		CASE FC OF
		(******************************************************************)
		1..2: (* 0x01 Read Coil Status , 0x02 Read Input Status *)
			IF R_POINTS <= 2000 THEN
				w_tmp := INT_TO_WORD(R_ADDR);
				S_BUF.BUFFER[08] := WORD_TO_BYTE(SHR(w_tmp,8));
				S_BUF.BUFFER[09] := WORD_TO_BYTE(w_tmp);
				w_tmp := INT_TO_WORD(R_POINTS);
				S_BUF.BUFFER[10] := WORD_TO_BYTE(SHR(w_tmp,8));
				S_BUF.BUFFER[11] := WORD_TO_BYTE(w_tmp);
				S_BUF.SIZE := UINT#12;
				Response :=	WORD_TO_INT(SHR(INT_TO_WORD(R_POINTS + 7),3));
				comp := 7;
			ELSE
				ERROR := DWORD#2; (* ILLEGAL DATA ADDRESS *)
			END_IF;
		(******************************************************************)
		3..4: (* 0x03 Read Holding Registers , 0x04 Read Input Registers *)
			IF R_POINTS <= 125 THEN
				w_tmp := INT_TO_WORD(R_ADDR);
				S_BUF.BUFFER[08] := WORD_TO_BYTE(SHR(w_tmp,8));
				S_BUF.BUFFER[09] := WORD_TO_BYTE(w_tmp);
				w_tmp := INT_TO_WORD(R_POINTS);
				S_BUF.BUFFER[10] := WORD_TO_BYTE(SHR(w_tmp,8));
				S_BUF.BUFFER[11] := WORD_TO_BYTE(w_tmp);
				S_BUF.SIZE := UINT#12;
				Response :=	WORD_TO_INT(SHL(w_tmp,1));
				comp := 7;
			ELSE
				ERROR := DWORD#2; (* ILLEGAL DATA ADDRESS *)
			END_IF;
		(******************************************************************)
		5:	(* 0x05 Force Single Coil *)
			IF W_DATA_ADR <= DATA_SIZE THEN
				w_tmp := INT_TO_WORD(W_ADDR);
				S_BUF.BUFFER[08] := WORD_TO_BYTE(SHR(w_tmp,8));
				S_BUF.BUFFER[09] := WORD_TO_BYTE(w_tmp);
				S_BUF.BUFFER[10] := SEL((DATA[W_DATA_ADR] AND SHL(WORD#1,W_DATA_BITPOS))>WORD#00,BYTE#16#00,BYTE#16#FF);
				S_BUF.BUFFER[11] := BYTE#00;
				S_BUF.SIZE := UINT#12;
				Response := 3;
				comp := 11;
			ELSE
				ERROR := DWORD#2; (* ILLEGAL DATA ADDRESS *)
			END_IF;
		(******************************************************************)
		6:	(* 0x06 Preset Single Register *)
			IF W_DATA_ADR <= DATA_SIZE THEN
				w_tmp := INT_TO_WORD(W_ADDR);
				S_BUF.BUFFER[08] := WORD_TO_BYTE(SHR(w_tmp,8));
				S_BUF.BUFFER[09] := WORD_TO_BYTE(w_tmp);
				w_tmp := DATA[W_DATA_ADR];
				S_BUF.BUFFER[10] := WORD_TO_BYTE(SHR(w_tmp,8));
				S_BUF.BUFFER[11] := WORD_TO_BYTE(w_tmp);
				S_BUF.SIZE := UINT#12;
				Response := 3;
				comp := 11;
			ELSE
				ERROR := DWORD#2; (* ILLEGAL DATA ADDRESS *)
			END_IF;
		(******************************************************************)
		15:	(* 0x0F Force Multiple Coils *)
			IF (WORD_TO_INT(SHR(INT_TO_WORD(WORD_TO_INT(SHL(INT_TO_WORD(W_DATA_ADR),4)) + W_POINTS + W_DATA_BITPOS + 15),4)) <= DATA_SIZE) AND W_POINTS <= 1968 THEN
				w_tmp := INT_TO_WORD(W_ADDR);
				S_BUF.BUFFER[08] := WORD_TO_BYTE(SHR(w_tmp,8));
				S_BUF.BUFFER[09] := WORD_TO_BYTE(w_tmp);
				w_tmp := INT_TO_WORD(W_POINTS);
				S_BUF.BUFFER[10] := WORD_TO_BYTE(SHR(w_tmp,8));
				S_BUF.BUFFER[11] := WORD_TO_BYTE(w_tmp);
				S_BUF.BUFFER[12] := WORD_TO_BYTE(SHR(INT_TO_WORD(W_POINTS + 7),3));

				w_mask := SHL(WORD#1,W_DATA_BITPOS);
				bit_pos := 0;
				w_tmp := WORD#00;
				idx1 := 12;
				idx2 := W_DATA_ADR;
				FOR i := 1 TO W_POINTS DO
					w_tmp :=OSCAT_BASIC.BIT_LOAD_W(w_tmp,(DATA[idx2] AND w_mask) > WORD#0,bit_pos);
					bit_pos := bit_pos + 1;
					IF bit_pos > 7 OR i=W_POINTS THEN
						bit_pos := 0;
						idx1 := idx1 + 1;
						S_BUF.BUFFER[idx1] := WORD_TO_BYTE(w_tmp);
						w_tmp := WORD#0;
					END_IF;
					w_mask := ROL(w_mask,1);
					IF w_mask = WORD#1 THEN
						idx2 := idx2 +1;
					END_IF;
				END_FOR;
				S_BUF.SIZE := INT_TO_UINT(idx1 + 1);
				Response := 3;
				comp := 11;
			ELSE
				ERROR := DWORD#2; (* ILLEGAL DATA ADDRESS *)
			END_IF;
		(******************************************************************)
		16:	(* 0x10 Write Multiple Registers *)
			IF W_DATA_ADR + W_POINTS <= DATA_SIZE AND W_POINTS <= 123 THEN
				w_tmp := INT_TO_WORD(W_ADDR);
				S_BUF.BUFFER[08] := WORD_TO_BYTE(SHR(w_tmp,8));
				S_BUF.BUFFER[09] := WORD_TO_BYTE(w_tmp);
				w_tmp := INT_TO_WORD(W_POINTS);
				S_BUF.BUFFER[10] := WORD_TO_BYTE(SHR(w_tmp,8));
				S_BUF.BUFFER[11] := WORD_TO_BYTE(w_tmp);
				S_BUF.BUFFER[12] := SHL(S_BUF.BUFFER[11],1);
			
				idx1 := 11;
				count := W_DATA_ADR + W_POINTS - 1;
				FOR i := W_DATA_ADR TO count DO
					idx1 := idx1 + 2;
					idx2 := idx1 + 1; (* zweiter index für pcworx notwendig ! *)
					w_tmp := DATA[i];
					S_BUF.BUFFER[idx1] := WORD_TO_BYTE(SHR(w_tmp,8));
					S_BUF.BUFFER[idx2] := WORD_TO_BYTE(w_tmp);
				END_FOR;

				S_BUF.SIZE := INT_TO_UINT(idx2 + 1);
				Response := 3;
				comp := 11;
			ELSE
				ERROR := DWORD#2; (* ILLEGAL DATA ADDRESS *)
			END_IF;
		(******************************************************************)
		22:	(* 0x16 Mask Write Register *)
			IF W_DATA_ADR + 2 <= DATA_SIZE THEN
				w_tmp := INT_TO_WORD(W_ADDR);
				S_BUF.BUFFER[08] := WORD_TO_BYTE(SHR(w_tmp,8));
				S_BUF.BUFFER[09] := WORD_TO_BYTE(w_tmp);
				idx1 := W_DATA_ADR;
				w_tmp := DATA[idx1];
				S_BUF.BUFFER[10] := WORD_TO_BYTE(SHR(w_tmp,8));
				S_BUF.BUFFER[11] := WORD_TO_BYTE(w_tmp);
				idx1 := idx1 +1;
				w_tmp := DATA[idx1];
				S_BUF.BUFFER[12] := WORD_TO_BYTE(SHR(w_tmp,8));
				S_BUF.BUFFER[13] := WORD_TO_BYTE(w_tmp);

				S_BUF.SIZE := UINT#14;
				Response := 5;
				comp := 13;
			ELSE
				ERROR := DWORD#2; (* ILLEGAL DATA ADDRESS *)
			END_IF;
		(******************************************************************)
		23:	(* 0x17 Read/Write Multible Registers *)
			IF W_DATA_ADR + W_POINTS <= DATA_SIZE AND W_POINTS <= 121 AND R_POINTS <= 125 THEN
				idx1 := 15;
				count := W_DATA_ADR + W_POINTS - 1;
				FOR i := W_DATA_ADR TO count DO
					idx1 := idx1 + 2;
					idx2 := idx1 + 1; (* zweiter index für pcworx notwendig ! *)
					w_tmp := DATA[i];
					S_BUF.BUFFER[idx1] := WORD_TO_BYTE(SHR(w_tmp,8));
					S_BUF.BUFFER[idx2] := WORD_TO_BYTE(w_tmp);
				END_FOR;

				(* WRITE *)
				w_tmp := INT_TO_WORD(W_ADDR);
				S_BUF.BUFFER[12] := WORD_TO_BYTE(SHR(w_tmp,8));
				S_BUF.BUFFER[13] := WORD_TO_BYTE(w_tmp);
				w_tmp := INT_TO_WORD(W_POINTS);
				S_BUF.BUFFER[14] := WORD_TO_BYTE(SHR(w_tmp,8));
				S_BUF.BUFFER[15] := WORD_TO_BYTE(w_tmp);
				S_BUF.BUFFER[16] := SHL(S_BUF.BUFFER[15],1);

				(* READ *)
				w_tmp := INT_TO_WORD(R_ADDR);
				S_BUF.BUFFER[08] := WORD_TO_BYTE(SHR(w_tmp,8));
				S_BUF.BUFFER[09] := WORD_TO_BYTE(w_tmp);
				w_tmp := INT_TO_WORD(R_POINTS);
				S_BUF.BUFFER[10] := WORD_TO_BYTE(SHR(w_tmp,8));
				S_BUF.BUFFER[11] := WORD_TO_BYTE(w_tmp);

				S_BUF.SIZE := INT_TO_UINT(idx2 + 1);
				Response := WORD_TO_INT(SHL(w_tmp,1));
				comp := 7;
			ELSE
				ERROR := DWORD#2; (* ILLEGAL DATA ADDRESS *)
			END_IF;
		(******************************************************************)

		ELSE
			ERROR := DWORD#00000001; (* ILLEGAL FUNCTION *)
		END_CASE;

		(* Daten senden *)
		IF ERROR = DWORD#00 THEN
			Transaction_ID := Transaction_ID + 1;
			w_tmp := UINT_TO_WORD(S_BUF.SIZE - UINT#6);
			(* ---- H E A D E R --------------------------------------------------------------- *)
			S_BUF.BUFFER[0] := IP_ID; (* TRANSACTION-ID HI-Byte *)
			S_BUF.BUFFER[1] := INT_TO_BYTE(Transaction_ID); (* TRANSACTION-ID LO-Byte *)
			S_BUF.BUFFER[2] := BYTE#00; (* PROTOKOLL-ID HI-Byte *)
			S_BUF.BUFFER[3] := BYTE#00; (* PROTOKOLL-ID LO-Byte *)
			S_BUF.BUFFER[4] := WORD_TO_BYTE(SHR(w_tmp,8)); (* Laenge HI-Byte *)
			S_BUF.BUFFER[5] := WORD_TO_BYTE(w_tmp); (* Laenge LO-Byte *)
			S_BUF.BUFFER[6] := UNIT_ID; (* UNIT *)
			S_BUF.BUFFER[7] := INT_TO_BYTE(FC); (* FUNCTION-CODE *)
			(*----- END OF HEADER --------------------------------------------------------------*)
			R_BUF.SIZE := UINT#0; (* Empfangsbuffer löschen *)
			state := 30; (* wait for response *)
		ELSE
			IP_STATE := BYTE#4; (* Abmelden *)
			state := 00;
		END_IF;
	END_IF;

30: (* response *)
	IF IP_C.ERROR <> DWORD#00 THEN
		ERROR := IP_C.ERROR;
		IP_STATE := BYTE#4; (* Abmelden *)
		state := 00;
	ELSIF S_BUF.SIZE = UINT#0 AND R_BUF.SIZE > UINT#0 THEN
		(* erwartete länge in sendebuffer nachträglich eintragen um vergleich zu ermöglichen *)
		w_tmp := INT_TO_WORD(Response + 3);
		S_BUF.BUFFER[4] := WORD_TO_BYTE(SHR(w_tmp,8));
		S_BUF.BUFFER[5] := WORD_TO_BYTE(w_tmp);

		FOR i := 0 TO comp DO
			IF S_BUF.BUFFER[i] <> R_BUF.BUFFER[i] THEN EXIT; END_IF;
		END_FOR;

		IF R_BUF.SIZE >= UINT#9 AND R_BUF.BUFFER[7] > BYTE#128 THEN  (* Bit 7 = Error Message *)
			ERROR := BYTE_TO_DWORD(R_BUF.BUFFER[8]);
			IP_STATE := BYTE#4; (* Abmelden *)
			state := 00;
		ELSIF R_BUF.SIZE = INT_TO_UINT(Response + 9) AND i > comp THEN
			mask := SHL(DWORD#1,FC);
			(* READ_COILS, READ_INPUT_DISCRETES *)
			IF (mask AND DWORD#2#00000000_00000000_00000000_00000110) > DWORD#0 THEN (* FC 1,2 *)
				IF WORD_TO_INT(SHR(INT_TO_WORD(WORD_TO_INT(SHL(INT_TO_WORD(R_DATA_ADR),4)) + R_POINTS + R_DATA_BITPOS + 15),4)) <= DATA_SIZE THEN
					b_mask := BYTE#1;
					idx1 := 09;
					idx2 := R_DATA_ADR;
					bit_pos := R_DATA_BITPOS;
					FOR i := 1 TO R_POINTS DO
						DATA[idx2]:=OSCAT_BASIC.BIT_LOAD_W(DATA[idx2],(R_BUF.BUFFER[idx1] AND b_mask) > BYTE#0,bit_pos);
						bit_pos := bit_pos + 1;
						IF bit_pos > 15 THEN
							idx2 := idx2 + 1;
							bit_pos := 0;
						END_IF;
						b_mask := ROL(b_mask,1);
						IF b_mask = BYTE#1 THEN
							idx1 := idx1 + 1;
						END_IF;
					END_FOR;
				ELSE
					ERROR := DWORD#2; (* ILLEGAL DATA ADDRESS *)
				END_IF;

			(* READ_MULTIPLE_REGISTERS, READ_INPUT_REGISTERS, READ_WRITE_REGISTERS *)
			ELSIF (mask AND DWORD#2#00000000_10000000_00000000_00011000) > DWORD#0 THEN (* FC 3,4,23 *)
				IF R_DATA_ADR + R_POINTS <= DATA_SIZE THEN
					stop := R_DATA_ADR + R_POINTS -1 ;
					idx1 := 07;
					FOR i := R_DATA_ADR TO stop DO
						idx1 := idx1 + 2;
						idx2 := idx1 + 1;
						DATA[i] := OSCAT_BASIC.WORD_OF_BYTE(R_BUF.BUFFER[idx1],R_BUF.BUFFER[idx2]);
					END_FOR;
				ELSE
					ERROR := DWORD#2; (* ILLEGAL DATA ADDRESS *)
				END_IF;
			ELSIF (mask AND DWORD#2#11111111_00111110_01111111_10000001) > DWORD#0 THEN (* ILLEGAL FUNCTION CODE ? *)
				ERROR := DWORD#1; (* ILLEGAL FUNCTION *)
			END_IF;
		ELSE
			ERROR := DWORD#3; (* ILLEGAL DATA VALUE *)
		END_IF;

		IP_STATE := BYTE#4; (* Abmelden *)
		state := 00;
		R_BUF.SIZE := UINT#0;

	END_IF;

END_CASE;

(* IP_FIFO *)
IP_FIFO(FIFO:=IP_C.FIFO,STATE:=IP_STATE,ID:=IP_ID);
BUSY := IP_STATE = BYTE#3;

(* revision history
ks	05. jan. 2009	rev 1.0
	original version

ks	28. jan. 2009	rev 1.1
	network_buffer_short verwendet  

ks	20. oct. 2009	rev 1.2
Networkbuffer und Buffer-funktionen auf Basis 0

*)

END_FUNCTION_BLOCK

// POUs/NETWORK/MB_SERVER
FUNCTION_BLOCK MB_SERVER
VAR_IN_OUT
	IP_C : IP_C;
	S_BUF : NETWORK_BUFFER_SHORT;
	R_BUF : NETWORK_BUFFER_SHORT;
	VMAP : ARRAY [1..10] OF VMAP_DATA;
	DATA : ARRAY [0..255] OF WORD;
END_VAR
VAR_INPUT
	DATA_SIZE : INT;
	ENABLE : BOOL;
	UDP : BOOL;
END_VAR
VAR_OUTPUT
	ERROR : DWORD;
END_VAR
VAR
	MB_VMAP : MB_VMAP;
	adr1 : INT;
	adr2 : INT;
	points : INT;
	points2 : INT;
	coils : BYTE;
	mask : BYTE;
	idx1 : INT;
	idx2 : INT;
	bit_pos : INT;
	count : INT;
	fc : INT;
	i : INT;
	state : INT;
	ip_state : BYTE;
	ip_id : BYTE;
	IP_FIFO : IP_FIFO;
	w_tmp : WORD;
	last_cycle : TIME;
	tx : TIME;
	t : TON;
	ip_error : BOOL;
END_VAR

(*

version 1.4		05. may. 2012
programmer 		ks
tested by		ks

MB_SERVER ermöglicht das Lesen/Schreiben von Daten durch ein Remote-Device mittels Modbus over Ethernet (OpenModbus)

*)

(* read system time *)
tx := DWORD_TO_TIME(OSCAT_BASIC.T_PLC_MS());

FOR i := 1 TO 10 DO
	IF VMAP[i].TIME_OUT > T#0s THEN
		VMAP[i].TIME_OUT := VMAP[i].TIME_OUT + tx - last_cycle;
	END_IF;
END_FOR;
last_cycle := tx;
ip_error := IP_C.ERROR > DWORD#0;

CASE state OF
00: (* Warten auf Freigabe *)
	IF ENABLE THEN
		state := 10;
		ip_state := BYTE#1; (* Anmelden *)
	END_IF;

10: (* Bei IP_Control anmelden und auf freigabe warten *)
	IF ip_state = BYTE#3 THEN

		(* IP Datenverkehr einrichten *)
		IP_C.C_PORT := WORD#0; (* Port von IP_CONTROL verwenden *)
		IP_C.C_IP := DWORD#0; (* IP von IP_CONTROL verwenden *)
		IP_C.C_MODE := SEL(UDP,BYTE#4,BYTE#5); (* Mode: 4=TCP+PASSIV+PORT , 5=UDP+PASSIV+PORT *)
		IP_C.TIME_RESET := TRUE; (* Zeitueberwachung rücksetzen *)
		IP_C.C_ENABLE := TRUE; (* Verbindungsaufbau freigeben *)
		IP_C.R_OBSERVE := TRUE; (* keine Empfangsueberwachung *)
		state := 20;
	END_IF;

20:	IF NOT ip_error THEN
		IF S_BUF.SIZE = UINT#0 AND R_BUF.SIZE > UINT#6 THEN	(* Datensenden nicht aktiv und Daten wurden empfangen *)
			IF  R_BUF.SIZE = WORD_TO_UINT(OSCAT_BASIC.WORD_OF_BYTE(R_BUF.BUFFER[4],R_BUF.BUFFER[5])) + UINT#6 THEN (* gültige Datenlänge *)
				ERROR := DWORD#00; (* Error löschen *)

				(* Header kopieren *)
				FOR i := 0 TO 13 DO
					S_BUF.BUFFER[i] := R_BUF.BUFFER[i];
				END_FOR;
				fc := BYTE_TO_INT(R_BUF.BUFFER[7]);
				adr1 := WORD_TO_INT(OSCAT_BASIC.WORD_OF_BYTE(R_BUF.BUFFER[8],R_BUF.BUFFER[9]));
				points := WORD_TO_INT(OSCAT_BASIC.WORD_OF_BYTE(R_BUF.BUFFER[10],R_BUF.BUFFER[11]));

				(* Virtual Address *)
				MB_VMAP(VMAP:=VMAP,FC:=fc,V_ADR:=adr1,V_CNT:=points,SIZE:=DATA_SIZE);
				adr1:=MB_VMAP.P_ADR;
				bit_pos:=MB_VMAP.P_BIT;
				ERROR:=BYTE_TO_DWORD(MB_VMAP.ERROR);

				IF ERROR = DWORD#0 THEN
					CASE fc OF
					(*---------------------------------------------*)
					1..2 : (* Read Coil Status / Read Input Status *)
						count := 9; (* erstes Datenbyte *)
						coils := BYTE#0;
						mask := BYTE#1;
						FOR i := 1 TO points DO
							IF mask = BYTE#0 THEN
								mask := BYTE#1;
								S_BUF.BUFFER[count] := coils;
								coils := BYTE#0;
								count := count + 1;
							END_IF;
							IF (DATA[adr1] AND SHL(WORD#1,bit_pos)) > WORD#0 THEN
								coils := coils OR mask;
							END_IF;
	
							bit_Pos := bit_Pos + 1;
							IF bit_pos > 15 THEN
								ADR1 := ADR1 + 1;
								bit_pos := 0;
							END_IF;
	
							mask := SHL(mask,1);
						END_FOR;
						S_BUF.BUFFER[Count] := coils;
	
						S_BUF.BUFFER[8] := INT_TO_BYTE(count - 8); (* Bytecount *)
						S_BUF.SIZE := INT_TO_UINT(count + 1);
	
					(*--------------------------------------------------*)
					3..4 : (* Read Holding Registers / Read Input Registers *)
						idx1 := 07;
						count := adr1 + points - 1;
						FOR i := adr1 TO count DO
							idx1 := idx1 + 2;
							idx2 := idx1 + 1; (* zweiter index für pcworx notwendig ! *)
							w_tmp := DATA[i];
							S_BUF.BUFFER[idx1] := WORD_TO_BYTE(SHR(w_tmp,8));
							S_BUF.BUFFER[idx2] := WORD_TO_BYTE(w_tmp);
						END_FOR;
						S_BUF.BUFFER[8] := SHL(INT_TO_BYTE(points),1); (* Anzahl Register in Bytes *)
						S_BUF.SIZE := INT_TO_UINT(idx2 + 1);
					(*--------------------------------------------------*)
					5 : (* Force Single Coil *)
						DATA[adr1]:=OSCAT_BASIC.BIT_LOAD_W(DATA[adr1],R_BUF.BUFFER[10] > BYTE#0,bit_pos);
						S_BUF.SIZE := UINT#12;
					(*--------------------------------------------------*)
					6 : (* Preset Single Register *)
						DATA[adr1] := OSCAT_BASIC.WORD_OF_BYTE(R_BUF.BUFFER[10],R_BUF.BUFFER[11]);
						S_BUF.SIZE := UINT#12;
					(*--------------------------------------------------*)
					15 : (* Force Multible Coils *)
						mask := BYTE#1;
						idx1 := 13;
						FOR i := 1 TO points DO
							DATA[adr1]:=OSCAT_BASIC.BIT_LOAD_W(DATA[adr1],(R_BUF.BUFFER[idx1] AND mask) > BYTE#0,bit_pos);
							bit_pos := bit_pos + 1;
							IF bit_pos > 15 THEN
								adr1:= adr1 + 1;
								bit_pos := 0;
							END_IF;
							mask := ROL(mask,1);
							IF mask = BYTE#1 THEN
								idx1 := idx1 +1;
							END_IF;
						END_FOR;
						S_BUF.SIZE := UINT#12;
					(*--------------------------------------------------*)
					16 : (* Preset Multiple Registers	*)
						idx1 := 11;
						count := adr1 + points - 1;
						FOR i := adr1 TO Count DO
							idx1 := idx1 + 2;
	 						idx2 := idx1 + 1;
							Data[i] := OSCAT_BASIC.WORD_OF_BYTE(R_BUF.BUFFER[idx1],R_BUF.BUFFER[idx2]);
						END_FOR;
						S_BUF.SIZE := UINT#12;
					(*--------------------------------------------------*)
					22 : (* Mask Write Register *)
						w_tmp := OSCAT_BASIC.WORD_OF_BYTE(R_BUF.BUFFER[10],R_BUF.BUFFER[11]); (* and mask *)
						DATA[adr1] := (DATA[adr1] AND w_tmp) OR (OSCAT_BASIC.WORD_OF_BYTE(R_BUF.BUFFER[12],R_BUF.BUFFER[13]) AND (NOT w_tmp));
						S_BUF.SIZE := UINT#14;
					(*--------------------------------------------------*)
					23 : (* Read / Write Registers	*)
						(*--- Write-Register -----------------------------------*)
						adr2 := WORD_TO_INT(OSCAT_BASIC.WORD_OF_BYTE(R_BUF.BUFFER[12],R_BUF.BUFFER[13]));
						points2 := WORD_TO_INT(OSCAT_BASIC.WORD_OF_BYTE(R_BUF.BUFFER[14],R_BUF.BUFFER[15]));

						(* Virtual Address Write Register *)
						MB_VMAP(VMAP:=VMAP,FC:=16,V_ADR:=adr2,V_CNT:=points2,SIZE:=DATA_SIZE);
						adr2:=MB_VMAP.P_ADR;
						ERROR:=BYTE_TO_DWORD(MB_VMAP.ERROR);
	
						IF ERROR = DWORD#0 THEN
							idx1 := 15;
							count := adr2 + points2 - 1;
							FOR i := adr2 TO count DO
								idx1 := idx1 + 2;
	 							idx2 := idx1 + 1; (* zweiter index für pcworx notwendig ! *)
								Data[i] := OSCAT_BASIC.WORD_OF_BYTE(R_BUF.BUFFER[idx1],R_BUF.BUFFER[idx2]);
							END_FOR;
	
							(*--- Read-Register -----------------------------------*)
							idx1 := 07;
							count := adr1 + points - 1;
							FOR i := adr1 TO count DO
								idx1 := idx1 + 2;
								idx2 := idx1 + 1; (* zweiter index für pcworx notwendig ! *)
								w_tmp := DATA[i];
								S_BUF.BUFFER[idx1] := WORD_TO_BYTE(SHR(w_tmp,8));
								S_BUF.BUFFER[idx2] := WORD_TO_BYTE(w_tmp);
							END_FOR;
							S_BUF.BUFFER[8] := SHL(INT_TO_BYTE(points),1); (* Anzahl Register in Bytes *)
							S_BUF.SIZE := INT_TO_UINT(idx2 + 1);
	
						END_IF;
	
					(*--------------------------------------------------*)
					ELSE
						ERROR := DWORD#01; (* ILLEGAL FUNCTION *)
					END_CASE;
				END_IF;
			END_IF;
	
			IF ERROR > DWORD#0 THEN
				S_BUF.BUFFER[7] := S_BUF.BUFFER[7] OR BYTE#2#1000_0000; (* Fehlerbit setzen *)
				S_BUF.BUFFER[8] := DWORD_TO_BYTE(ERROR);
				S_BUF.SIZE := UINT#9;
			END_IF;
	
			S_BUF.BUFFER[4] := BYTE#0; (* high Byte *)
			S_BUF.BUFFER[5] := UINT_TO_BYTE(S_BUF.SIZE - UINT#6); (* Längenfeld eintragen - nur low byte *)
	
		END_IF;
	ELSE
		ERROR := IP_C.ERROR;
	END_IF;

	t(IN:= ip_error, PT:=T#2s);
	IF t.Q THEN
		IP_C.TIME_RESET := TRUE; (* Error Reset *)
	END_IF;

	R_BUF.SIZE := UINT#0; (* Empfangsdaten zerstören *)

	IF ENABLE = FALSE OR t.Q THEN
	    ip_state := BYTE#4; (* Abmelden *)
		state := 00;
		IP_C.C_ENABLE := FALSE;
	END_IF;
END_CASE;

(* IP_FIFO *)
IP_FIFO(FIFO:=IP_C.FIFO,STATE:=ip_state,ID:=ip_id);

(* revision history
ks	05. jan. 2009	rev 1.0
	original version

ks	28. jan. 2009	rev 1.1
	network_buffer_short verwendet  

ks	20. oct. 2009	rev 1.2
	change lokal-var adr to adr1,Networkbuffer und Buffer-funktionen auf Basis 0

ks	17. may. 2011	rev 1.3
	automatischer re-connect

ks	05. may. 2012	rev 1.4
	timeoutüberwachung für re-connect
*)

END_FUNCTION_BLOCK

// POUs/NETWORK/MB_VMAP
FUNCTION_BLOCK MB_VMAP
VAR_IN_OUT
	VMAP :  ARRAY [1..10] OF VMAP_DATA;
END_VAR
VAR_INPUT
	FC : INT;
	V_ADR : INT;
	V_CNT : INT;
	SIZE : INT;
END_VAR
VAR_OUTPUT
	P_ADR : INT;
	P_BIT : INT;
	ERROR : BYTE;
END_VAR
VAR
	i : INT;
	vopt : DWORD;
	vadr : INT;
	padr : INT;
	mask : DWORD;
	vsize : INT;
	w_tmp : WORD;
	i_tmp : INT;
	init : BOOL;
END_VAR

(*
version 1.1		20. oct. 2009
programmer 		ks
tested by		ks

MB_VMAP Virtuelles Adress-Mapping für MB_SERVER
*)

IF init = FALSE THEN
	init := TRUE;
	IF VMAP[1].FC = DWORD#0 THEN
		VMAP[1].FC := DWORD#16#FFFF_FFFF;
		VMAP[1].V_ADR := 0;
		VMAP[1].V_SIZE := 256;
		VMAP[1].P_ADR := 0;
	END_IF;
END_IF;

ERROR := BYTE#02; (* ILLEGAL DATA ADDRESS *)
mask := SHL(DWORD#1,FC);

IF (mask AND DWORD#2#00000000_01000000_00000000_01100000) <> DWORD#0 THEN (* FC 5,6,22 *)
	V_CNT := 1;
ELSIF V_CNT = 0 THEN
	RETURN;
END_IF;

FOR i := 1 TO 10 DO
	vopt := VMAP[i].FC; 
	IF (vopt AND mask) <> DWORD#0 THEN
		vadr := VMAP[i].V_ADR;
		vsize := VMAP[i].V_SIZE;
		padr := VMAP[i].P_ADR;

		IF (mask AND DWORD#2#00000000_00000000_10000000_00100110) <> DWORD#0 THEN (* FC 1,2,5,15 für Bit-Access *)
			i_tmp := WORD_TO_INT(SHR(INT_TO_WORD(V_ADR + V_CNT -1),4))+1;
			IF i_tmp <= SIZE AND i_tmp <= vsize THEN
				w_tmp := INT_TO_WORD(V_ADR);
				P_ADR := WORD_TO_INT(SHR(w_tmp,4)) + padr; 
				P_BIT := WORD_TO_INT(w_tmp AND WORD#16#000F);
				ERROR := BYTE#0;
				EXIT;
			END_IF;
		ELSIF (mask AND DWORD#2#00000000_11000001_00000000_01011000) <> DWORD#0 THEN (* FC 3,4,6,16,22,23 für Register-Access *)
			IF V_ADR >= vadr AND V_ADR + V_CNT <= vadr + vsize THEN (* gültiger virtueller bereich *)
				P_ADR := V_ADR - vadr + padr; (* reale Adresse berechnen *)
				IF P_ADR + V_CNT <= SIZE THEN (* bereichsueberschreitung ? *)
					ERROR := BYTE#0;
					EXIT;
				END_IF;
			END_IF;
		ELSE
			ERROR := BYTE#01; (* ILLEGAL FUNCTION *)
			RETURN;
		END_IF;
	END_IF;
END_FOR;

IF ERROR = BYTE#0 THEN
	IF (mask AND DWORD#2#00000000_11000001_10000000_01100000) <> DWORD#0 THEN (* FC 5,6,15,16,22,23 Schreib-zugriff *)
		VMAP[i].TIME_OUT := T#1ms;
	END_IF;
END_IF;

(* revision history
ks	05. jan. 2009	rev 1.0
	original version

ks	20. oct. 2009	rev 1.1
	fehlerkorrektur in bitmaske

*)

END_FUNCTION_BLOCK

// POUs/NETWORK/MB_SERVER_1
FUNCTION_BLOCK MB_SERVER_1
VAR_IN_OUT
	IP_C : IP_C;
	S_BUF : NETWORK_BUFFER_SHORT;
	R_BUF : NETWORK_BUFFER_SHORT;
	VMAP : ARRAY [1..10] OF VMAP_DATA;
	DATA : ARRAY [0..255] OF WORD;
END_VAR
VAR_INPUT
	DATA_SIZE : INT;
	ENABLE : BOOL;
	UDP : BOOL;
END_VAR
VAR_OUTPUT
	ERROR : DWORD;
END_VAR
VAR
	MB_VMAP : MB_VMAP;
	adr1 : INT;
	adr2 : INT;
	points : INT;
	points2 : INT;
	coils : BYTE;
	mask : BYTE;
	idx1 : INT;
	idx2 : INT;
	bit_pos : INT;
	count : INT;
	fc : INT;
	i : INT;
	state : INT;
	ip_state : BYTE;
	ip_id : BYTE;
	IP_FIFO : IP_FIFO;
	w_tmp : WORD;
	last_cycle : TIME;
	tx : TIME;
	t : TON;
	ip_error : BOOL;
END_VAR

(*

version 1.3		17. may. 2011
programmer 		ks
tested by			ks

MB_SERVER ermöglicht das Lesen/Schreiben von Daten durch ein Remote-Device mittels Modbus over Ethernet (OpenModbus)

*)

(* read system time *)
tx := DWORD_TO_TIME(OSCAT_BASIC.T_PLC_MS());

FOR i := 1 TO 10 DO
	IF VMAP[i].TIME_OUT > T#0s THEN
		VMAP[i].TIME_OUT := VMAP[i].TIME_OUT + tx - last_cycle;
	END_IF;
END_FOR;
last_cycle := tx;
ip_error := IP_C.ERROR > DWORD#0;

CASE state OF
00: (* Warten auf Freigabe *)
	IF ENABLE THEN
		state := 10;
		ip_state := BYTE#1; (* Anmelden *)
	END_IF;

10: (* Bei IP_Control anmelden und auf freigabe warten *)
	IF ip_state = BYTE#3 THEN

		(* IP Datenverkehr einrichten *)
		IP_C.C_PORT := WORD#0; (* Port von IP_CONTROL verwenden *)
		IP_C.C_IP := DWORD#0; (* IP von IP_CONTROL verwenden *)
		IP_C.C_MODE := SEL(UDP,BYTE#4,BYTE#5); (* Mode: 4=TCP+PASSIV+PORT , 5=UDP+PASSIV+PORT *)
		IP_C.TIME_RESET := TRUE; (* Zeitueberwachung rücksetzen *)
		IP_C.C_ENABLE := TRUE; (* Verbindungsaufbau freigeben *)
		IP_C.R_OBSERVE := FALSE; (* keine Empfangsueberwachung *)
		state := 20;
	END_IF;

20:	IF NOT ip_error THEN
		IF S_BUF.SIZE = UINT#0 AND R_BUF.SIZE > UINT#6 THEN	(* Datensenden nicht aktiv und Daten wurden empfangen *)
			IF  R_BUF.SIZE = WORD_TO_UINT(OSCAT_BASIC.WORD_OF_BYTE(R_BUF.BUFFER[4],R_BUF.BUFFER[5])) + UINT#6 THEN (* gültige Datenlänge *)
				ERROR := DWORD#00; (* Error löschen *)
	
				(* Header kopieren *)
				FOR i := 0 TO 13 DO
					S_BUF.BUFFER[i] := R_BUF.BUFFER[i];
				END_FOR;
				fc := BYTE_TO_INT(R_BUF.BUFFER[7]);
				adr1 := WORD_TO_INT(OSCAT_BASIC.WORD_OF_BYTE(R_BUF.BUFFER[8],R_BUF.BUFFER[9]));
				points := WORD_TO_INT(OSCAT_BASIC.WORD_OF_BYTE(R_BUF.BUFFER[10],R_BUF.BUFFER[11]));
	
				(* Virtual Address *)
				MB_VMAP(VMAP:=VMAP,FC:=fc,V_ADR:=adr1,V_CNT:=points,SIZE:=DATA_SIZE);
				adr1:=MB_VMAP.P_ADR;
				bit_pos:=MB_VMAP.P_BIT;
				ERROR:=BYTE_TO_DWORD(MB_VMAP.ERROR);
	
				IF ERROR = DWORD#0 THEN
					CASE fc OF
					(*---------------------------------------------*)
					1..2 : (* Read Coil Status / Read Input Status *)
						count := 9; (* erstes Datenbyte *)
						coils := BYTE#0;
						mask := BYTE#1;
						FOR i := 1 TO points DO
							IF mask = BYTE#0 THEN
								mask := BYTE#1;
								S_BUF.BUFFER[count] := coils;
								coils := BYTE#0;
								count := count + 1;
							END_IF;
							IF (DATA[adr1] AND SHL(WORD#1,bit_pos)) > WORD#0 THEN
								coils := coils OR mask;
							END_IF;
	
							bit_Pos := bit_Pos + 1;
							IF bit_pos > 15 THEN
								ADR1 := ADR1 + 1;
								bit_pos := 0;
							END_IF;
	
							mask := SHL(mask,1);
						END_FOR;
						S_BUF.BUFFER[Count] := coils;
	
						S_BUF.BUFFER[8] := INT_TO_BYTE(count - 8); (* Bytecount *)
						S_BUF.SIZE := INT_TO_UINT(count + 1);
	
					(*--------------------------------------------------*)
					3..4 : (* Read Holding Registers / Read Input Registers *)
						idx1 := 07;
						count := adr1 + points - 1;
						FOR i := adr1 TO count DO
							idx1 := idx1 + 2;
							idx2 := idx1 + 1; (* zweiter index für pcworx notwendig ! *)
							w_tmp := DATA[i];
							S_BUF.BUFFER[idx1] := WORD_TO_BYTE(SHR(w_tmp,8));
							S_BUF.BUFFER[idx2] := WORD_TO_BYTE(w_tmp);
						END_FOR;
						S_BUF.BUFFER[8] := SHL(INT_TO_BYTE(points),1); (* Anzahl Register in Bytes *)
						S_BUF.SIZE := INT_TO_UINT(idx2 + 1);
					(*--------------------------------------------------*)
					5 : (* Force Single Coil *)
						DATA[adr1]:=OSCAT_BASIC.BIT_LOAD_W(DATA[adr1],R_BUF.BUFFER[10] > BYTE#0,bit_pos);
						S_BUF.SIZE := UINT#12;
					(*--------------------------------------------------*)
					6 : (* Preset Single Register *)
						DATA[adr1] := OSCAT_BASIC.WORD_OF_BYTE(R_BUF.BUFFER[10],R_BUF.BUFFER[11]);
						S_BUF.SIZE := UINT#12;
					(*--------------------------------------------------*)
					15 : (* Force Multible Coils *)
						mask := BYTE#1;
						idx1 := 13;
						FOR i := 1 TO points DO
							DATA[adr1]:=OSCAT_BASIC.BIT_LOAD_W(DATA[adr1],(R_BUF.BUFFER[idx1] AND mask) > BYTE#0,bit_pos);
							bit_pos := bit_pos + 1;
							IF bit_pos > 15 THEN
								adr1:= adr1 + 1;
								bit_pos := 0;
							END_IF;
							mask := ROL(mask,1);
							IF mask = BYTE#1 THEN
								idx1 := idx1 +1;
							END_IF;
						END_FOR;
						S_BUF.SIZE := UINT#12;
					(*--------------------------------------------------*)
					16 : (* Preset Multiple Registers	*)
						idx1 := 11;
						count := adr1 + points - 1;
						FOR i := adr1 TO Count DO
							idx1 := idx1 + 2;
	 						idx2 := idx1 + 1;
							Data[i] := OSCAT_BASIC.WORD_OF_BYTE(R_BUF.BUFFER[idx1],R_BUF.BUFFER[idx2]);
						END_FOR;
						S_BUF.SIZE := UINT#12;
					(*--------------------------------------------------*)
					22 : (* Mask Write Register *)
						w_tmp := OSCAT_BASIC.WORD_OF_BYTE(R_BUF.BUFFER[10],R_BUF.BUFFER[11]); (* and mask *)
						DATA[adr1] := (DATA[adr1] AND w_tmp) OR (OSCAT_BASIC.WORD_OF_BYTE(R_BUF.BUFFER[12],R_BUF.BUFFER[13]) AND (NOT w_tmp));
						S_BUF.SIZE := UINT#14;
					(*--------------------------------------------------*)
					23 : (* Read / Write Registers	*)
						(*--- Write-Register -----------------------------------*)
						adr2 := WORD_TO_INT(OSCAT_BASIC.WORD_OF_BYTE(R_BUF.BUFFER[12],R_BUF.BUFFER[13]));
						points2 := WORD_TO_INT(OSCAT_BASIC.WORD_OF_BYTE(R_BUF.BUFFER[14],R_BUF.BUFFER[15]));
	
						(* Virtual Address Write Register *)
						MB_VMAP(VMAP:=VMAP,FC:=16,V_ADR:=adr2,V_CNT:=points2,SIZE:=DATA_SIZE);
						adr2:=MB_VMAP.P_ADR;
						ERROR:=BYTE_TO_DWORD(MB_VMAP.ERROR);
	
						IF ERROR = DWORD#0 THEN
							idx1 := 15;
							count := adr2 + points2 - 1;
							FOR i := adr2 TO count DO
								idx1 := idx1 + 2;
	 							idx2 := idx1 + 1; (* zweiter index für pcworx notwendig ! *)
								Data[i] := OSCAT_BASIC.WORD_OF_BYTE(R_BUF.BUFFER[idx1],R_BUF.BUFFER[idx2]);
							END_FOR;
	
							(*--- Read-Register -----------------------------------*)
							idx1 := 07;
							count := adr1 + points - 1;
							FOR i := adr1 TO count DO
								idx1 := idx1 + 2;
								idx2 := idx1 + 1; (* zweiter index für pcworx notwendig ! *)
								w_tmp := DATA[i];
								S_BUF.BUFFER[idx1] := WORD_TO_BYTE(SHR(w_tmp,8));
								S_BUF.BUFFER[idx2] := WORD_TO_BYTE(w_tmp);
							END_FOR;
							S_BUF.BUFFER[8] := SHL(INT_TO_BYTE(points),1); (* Anzahl Register in Bytes *)
							S_BUF.SIZE := INT_TO_UINT(idx2 + 1);
	
						END_IF;
	
					(*--------------------------------------------------*)
					ELSE
						ERROR := DWORD#01; (* ILLEGAL FUNCTION *)
					END_CASE;
				END_IF;
			END_IF;
	
			IF ERROR > DWORD#0 THEN
				S_BUF.BUFFER[7] := S_BUF.BUFFER[7] OR BYTE#2#1000_0000; (* Fehlerbit setzen *)
				S_BUF.BUFFER[8] := DWORD_TO_BYTE(ERROR);
				S_BUF.SIZE := UINT#9;
			END_IF;
	
			S_BUF.BUFFER[4] := BYTE#0; (* high Byte *)
			S_BUF.BUFFER[5] := UINT_TO_BYTE(S_BUF.SIZE - UINT#6); (* Längenfeld eintragen - nur low byte *)
	
		END_IF;
	ELSE
		ERROR := IP_C.ERROR;
	END_IF;

	t(IN:= ip_error, PT:=T#5s);
	IF t.Q THEN
		IP_C.TIME_RESET := TRUE; (* Error Reset *)
	END_IF;

	R_BUF.SIZE := UINT#0; (* Empfangsdaten zerstören *)

	IF ENABLE = FALSE THEN
	    ip_state := BYTE#4; (* Abmelden *)
		state := 00;
	END_IF;
END_CASE;

(* IP_FIFO *)
IP_FIFO(FIFO:=IP_C.FIFO,STATE:=ip_state,ID:=ip_id);

(* revision history
ks	05. jan. 2009	rev 1.0
	original version

ks	28. jan. 2009	rev 1.1
	network_buffer_short verwendet  

ks	20. oct. 2009	rev 1.2
	change lokal-var adr to adr1,Networkbuffer und Buffer-funktionen auf Basis 0

ks	17. may. 2011	rev 1.3
	automatischer re-connect
*)

END_FUNCTION_BLOCK

// POUs/CONVERT/MD5_STR
FUNCTION_BLOCK MD5_STR
VAR_INPUT
	RUN: BOOL;
END_VAR
VAR_OUTPUT
	DONE: BOOL;
END_VAR
VAR_IN_OUT
	STR: STRING(OSCAT_BASIC.STRING_LENGTH);
	MD5 : ARRAY [0..15] OF BYTE;
END_VAR
VAR
	run_last: BOOL;
	MD5_STREAM : MD5_STREAM;
	buf : ARRAY [0..63] OF BYTE;
	mode : INT;
	size : UDINT;
	pos : UDINT;
END_VAR

(*
version 1.0	06. dec. 2009
programmer 	ks
tested BY	ks

MD5_STR berechnet den MD5 Hash eines Strings
*)

CASE mode OF
0:	(* Wait für Start *)
	IF RUN AND NOT run_last THEN
		DONE := FALSE;
		mode := 1; (* Initialisierung *)
		size := LEN(STR);
	END_IF;

2:	(* Data copy and Calc *)
	IF size > 0 THEN
		OSCAT_BASIC._STRING_TO_BUFFER(STR:=MID(STR, UDINT_TO_INT(SIZE), UDINT_TO_INT(POS) + 1), POS:=0, PT:=ADR(buf), SIZE:=SIZEOF(buf));
	END_IF;

3:	DONE := TRUE;
	mode := 0; (* Stop *)

END_CASE;

IF mode > 0 THEN
	MD5_STREAM(SIZE:=size, MODE:=mode, BUF:=buf, MD5:=MD5, POS=>pos);
END_IF;

run_last := RUN;

(* revision history

ks	6. dec. 2009 rev 1.0
	original version

*)

END_FUNCTION_BLOCK

// POUs/WEATHER/MOON_PHASE
FUNCTION_BLOCK MOON_PHASE
VAR_INPUT
	XDT : DT;
	SCALE : BYTE := 12;
	UPDATE : TIME := T#1h;
END_VAR
VAR_OUTPUT
	PHASE : BYTE;
END_VAR
VAR
	x : UDINT;
	last_dt : DT;
END_VAR

(*
version 1.0		15. may. 2011
programmer		ks
tested by			ks

MOON_PHASE berechnet die aktuelle Mondphase
*)

IF XDT - last_dt > UPDATE THEN
	x := (DT_TO_UDINT(XDT) - 603240) MOD 2551392;
	PHASE := UDINT_TO_BYTE(SCALE * x / 2551392) ;
	last_dt := XDT;
END_IF;

(* revision history
ks	15.may. 2011	rev 1.0
	original version

*)

END_FUNCTION_BLOCK

// POUs/NET_VAR/NET_VAR_BOOL8
FUNCTION_BLOCK NET_VAR_BOOL8
VAR_IN_OUT
	X : NET_VAR_DATA;
END_VAR
VAR_INPUT
	IN1 : BOOL;
	IN2 : BOOL;
	IN3 : BOOL;
	IN4 : BOOL;
	IN5 : BOOL;
	IN6 : BOOL;
	IN7 : BOOL;
	IN8 : BOOL;
END_VAR
VAR_OUTPUT
	OUT1 : BOOL;
	OUT2 : BOOL;
	OUT3 : BOOL;
	OUT4 : BOOL;
	OUT5 : BOOL;
	OUT6 : BOOL;
	OUT7 : BOOL;
	OUT8 : BOOL;
	ID : BYTE;
END_VAR
VAR
	init : BOOL;
	index : INT;
	index2 : INT;
	BYTE_TO_BITS : OSCAT_BASIC.BYTE_TO_BITS;
END_VAR

(*
version 1.0		15. may. 2011
programmer		ks
tested by			ks

NET_VAR_BOOL8 überträgt bidirektional 8 boolsche Werte vom Master zum Client
*)

IF NOT init THEN
	init := TRUE;
	X.ID_MAX := X.ID_MAX + USINT#1;
	ID := USINT_TO_BYTE(X.ID_MAX);
END_IF;

IF X.STATE > BYTE#0 AND X.ERROR_ID = BYTE#0 THEN
	index := X.index; (* PCWORX Workaround *)
	IF INT_TO_UINT(index + 3) > X.BUF_SIZE THEN
		X.ERROR_ID := ID;
	ELSE
		IF X.STATE = BYTE#1 THEN (* Daten schreiben *)
			X.S_BUF.BUFFER[index] := ID; (* ID *)
			index := index + 1;
			X.S_BUF.BUFFER[index] := BYTE#4; (* TYPE BOOL8 *)
			index := index + 1;
			X.S_BUF.BUFFER[index] := OSCAT_BASIC.BYTE_OF_BIT(IN1,IN2,IN3,IN4,IN5,IN6,IN7,IN8);
			index := index + 1;

		ELSIF X.STATE = BYTE#2 THEN (* Daten lesen *)
			index2 := index + 1; (* PCWORX Workaround *)
			IF X.R_BUF.BUFFER[index] <> ID OR X.R_BUF.BUFFER[index2] <> BYTE#4 THEN
				X.ERROR_ID := ID;
			ELSE
				index := index + 2;
				BYTE_TO_BITS(IN:=X.R_BUF.BUFFER[index]);
				OUT1 := BYTE_TO_BITS.B0;
				OUT2 := BYTE_TO_BITS.B1;
				OUT3 := BYTE_TO_BITS.B2;
				OUT4 := BYTE_TO_BITS.B3;
				OUT5 := BYTE_TO_BITS.B4;
				OUT6 := BYTE_TO_BITS.B5;
				OUT7 := BYTE_TO_BITS.B6;
				OUT8 := BYTE_TO_BITS.B7;
				index := index + 1;
			END_IF;
		END_IF;
		X.index := index;
	END_IF;
END_IF;

(* revision history
ks	15.may. 2011	rev 1.0
	original version

*)

END_FUNCTION_BLOCK

// POUs/NET_VAR/NET_VAR_BUFFER
FUNCTION_BLOCK NET_VAR_BUFFER
VAR_IN_OUT
	BUF_IN : ARRAY[1..64] OF BYTE;
	BUF_OUT : ARRAY[1..64] OF BYTE;
	X : NET_VAR_DATA;
END_VAR
VAR_OUTPUT
	ID : BYTE;
END_VAR
VAR
	size : INT;
	init : BOOL;
	index : INT;
	index2 : INT;
END_VAR

(*
version 1.0		15. may. 2011
programmer		ks
tested by			ks

NET_VAR_BUFFER überträgt bidirektional 64 Bytes vom Master zum Client
*)

IF NOT init THEN
	init := TRUE;
	X.ID_MAX := X.ID_MAX + USINT#1;
	ID := USINT_TO_BYTE(X.ID_MAX);
END_IF;

IF X.STATE > BYTE#0 AND X.ERROR_ID = BYTE#0 THEN
	index := X.index; (* PCWORX Workaround *)
	IF X.STATE = BYTE#1 THEN (* Daten schreiben *)
		size := SIZEOF(BUF_IN);
		IF INT_TO_UINT(index + 3 + size) > X.BUF_SIZE THEN
			X.ERROR_ID := ID;
		ELSE
			X.S_BUF.BUFFER[index] := ID; (* ID *)
			index := index + 1;
			X.S_BUF.BUFFER[index] := BYTE#20; (* TYPE BUFFER *)
			index := index + 1;
			X.S_BUF.BUFFER[index] := INT_TO_BYTE(size); (* Anzahl der Bytes *)
				index := index + 1;
			FOR index2 := 1 TO size DO
				X.S_BUF.BUFFER[index] := BUF_IN[index2];
				index := index + 1;
			END_FOR;
		END_IF;
	ELSIF X.STATE = BYTE#2 THEN (* Daten lesen *)
		index2 := index + 1; (* PCWORX Workaround *)
		IF X.R_BUF.BUFFER[index] <> ID OR X.R_BUF.BUFFER[index2] <> BYTE#20 THEN
			X.ERROR_ID := ID;
		ELSE
			index := index + 2;
			size := BYTE_TO_INT(X.R_BUF.BUFFER[index]);
			index := index + 1;
			FOR index2 := 1 TO size DO
				BUF_OUT[index2] := X.R_BUF.BUFFER[index];
				index := index + 1;
			END_FOR;
		END_IF;
	END_IF;
	X.index := index;
END_IF;

(* revision history
ks	15.may. 2011	rev 1.0
	original version

*)

END_FUNCTION_BLOCK

// POUs/NET_VAR/NET_VAR_CONTROL
FUNCTION_BLOCK NET_VAR_CONTROL
VAR_INPUT
	ACTIVATE : BOOL;
	MASTER : BOOL;
	UDP : BOOL;
	REMOTE_IP4 : DWORD;
	REMOTE_PORT : WORD := 10000;
	SCAN_TIME : TIME := T#1s;
	WATCHDOG : TIME := T#2s;
END_VAR
VAR_OUTPUT
	RUN : BOOL;
	ERROR : DWORD;
END_VAR
VAR_IN_OUT
	X : NET_VAR_DATA;
END_VAR
VAR
	IPC : IP_CONTROL_V2;
	IP_C : IP_C; (* IP_Control Verwaltungsstruktur *)
	step : INT;
	activate_last : BOOL;
	tscan : TON;
	reset : BOOL;
END_VAR

(*
version 1.0		15. may. 2011
programmer		ks
tested by			ks

NET_VAR_CONTROL überträgt Daten bidirektional vom Master zum Client
*)

(* Typ
001 = BYTE
002 = WORD
003 = DWORD
004 = BOOL (8x)
005 = REAL
006 = STRING
007 = UINT
008 = INT
009 = DINT
010 = UDINT
013 = DWORD (8x)
015 = REAL (8x)

020 = BUFFER
021 = MIX (REAL,DINT,UDINT,
*)

IF X.ERROR_ID > BYTE#0 THEN (* Schwere Fehler bei Variablenzuordnung vorhanden  !! *)
	X.STATE := BYTE#0;
	ERROR := BYTE_TO_DWORD(X.ERROR_ID);
	X.ERROR_ID := BYTE#0;
	step := 999;
END_IF;

CASE step OF

00:	IF ACTIVATE AND NOT activate_last OR reset THEN

        (*  TCP + MASTER = C_MODE 0 (TCP + ACTIVE + PORT + IP) *)
        (*  UDP + MASTER = C_MODE 1 (UDP + ACTIVE + PORT + IP) *)
        (*  TCP + SLAVE  = C_MODE 2 (TCP + PASSIV + PORT + IP) *)
        (*  UDP + SLAVE  = C_MODE 3 (UDP + PASSIV + PORT + IP) *)
	IF MASTER THEN
		IP_C.C_MODE := BYTE#0;
		step := 100;
	ELSE
		IP_C.C_MODE := BYTE#2;
		step := 200;
	END_IF;
        IF UDP THEN IP_C.C_MODE := IP_C.C_MODE OR BYTE#1; END_IF;
	  	IP_C.C_PORT := REMOTE_PORT; (* Portnummer eintragen *)
	  	IP_C.C_IP := REMOTE_IP4; (* IP eintragen *)
	  	IP_C.TIME_RESET := TRUE; (* Zeitueberwachung rücksetzen *)
	  	IP_C.C_ENABLE := TRUE; (* Verbindungsaufbau freigeben *)
	  	IP_C.R_OBSERVE := TRUE; (* Empfangsueberwachung *)
		X.S_BUF.SIZE := UINT#0;
		X.R_BUF.SIZE := UINT#0;
		X.CYCLE := UDINT#0;
		X.ERROR_ID := BYTE#0;
		reset := FALSE;
	END_IF;

(* ++++++++++++++++++++++++++++++++++++++++++++++ *)

100:IF IP_C.C_STATE > BYTE#127 THEN (* Verbindung vorhanden *)
		X.STATE := BYTE#1; (* Daten sammeln *)
		X.BUF_SIZE := SIZEOF(X.S_BUF.BUFFER);
		X.S_BUF.BUFFER[0] := UDINT_TO_BYTE(X.CYCLE);
		X.INDEX := 1;
		step := 110;
	END_IF;

110:X.STATE := BYTE#0;
	X.S_BUF.SIZE := INT_TO_UINT(X.INDEX); (* Datenlänge eintragen *)
	step := 120;

120:IF X.S_BUF.SIZE = UINT#0 AND X.R_BUF.SIZE >= UINT#1 THEN (* länge der empfangenen Daten prüfen *)
		X.STATE := BYTE#2; (* Daten ausgeben *)
		X.BUF_SIZE := X.R_BUF.SIZE;
		X.INDEX := 1;
		X.ERROR_ID := BYTE#0;
		X.CYCLE := X.CYCLE + UDINT#1;
		ERROR := DWORD#0; (* nach erfolgreichen Zyklus letzten Fehlercode löschen *)
		RUN := TRUE;
		step := 130;
	END_IF;

130:X.STATE := BYTE#0;
	X.R_BUF.SIZE := UINT#0;
	IF NOT ACTIVATE THEN
		step := 999; (* Beenden *)
	ELSIF tscan.Q THEN
		step := 100;
	END_IF;

(* ++++++++++++++++++++++++++++++++++++++++++++++ *)

200:IF X.R_BUF.SIZE >= UINT#1 THEN
		X.STATE := BYTE#2; (* Daten ausgeben *)
		X.BUF_SIZE := X.R_BUF.SIZE;
		X.INDEX := 1;
		step := 210;
	END_IF;

210:X.STATE := BYTE#1; (* Daten sammeln *)
	X.BUF_SIZE := SIZEOF(X.R_BUF.BUFFER);;
	X.S_BUF.BUFFER[0] := X.R_BUF.BUFFER[0]; (* Cycle übernehmen *)
	X.INDEX := 1;
	X.R_BUF.SIZE := UINT#0;
	step := 220;

220:X.STATE := BYTE#0;
	X.S_BUF.SIZE := INT_TO_UINT(X.INDEX); (* Datenlänge eintragen *)
	step := 230;

230:IF X.S_BUF.SIZE = UINT#0 THEN
		ERROR := DWORD#0; (* nach erfolgreichen Zyklus letzten Fehlercode löschen *)
		RUN := TRUE;
		IF NOT ACTIVATE THEN
			step := 999; (* Beenden *)
		ELSE
			step := 200;
		END_IF;
	END_IF;

999:IP_C.C_ENABLE := FALSE; (* Beenden *)
	RUN := FALSE;
	step := 0;

END_CASE;

(* ++++++++++++++++++++++++++++++++++++++++++++++ *)

IPC(IP:= DWORD#0, PORT:= WORD#0 , TIME_OUT:= WATCHDOG, IP_C:= IP_C, S_BUF:= X.S_BUF, R_BUF:= X.R_BUF);

IF IP_C.ERROR > DWORD#0 THEN
	ERROR := IP_C.ERROR;
	RUN := FALSE;
	reset := TRUE;
	step := 0;
END_IF;

ACTIVATE_LAST := ACTIVATE; (* letzten Status sichern zur Flankenerkennung *)
tscan(IN:= step <> 110 ,PT:=SCAN_TIME);

(* revision history
ks	15.may. 2011	rev 1.0
	original version

*)

END_FUNCTION_BLOCK

// POUs/NET_VAR/NET_VAR_DWORD8
FUNCTION_BLOCK NET_VAR_DWORD8
VAR_IN_OUT
	X : NET_VAR_DATA;
END_VAR
VAR_INPUT
	IN1 : DWORD;
	IN2 : DWORD;
	IN3 : DWORD;
	IN4 : DWORD;
	IN5 : DWORD;
	IN6 : DWORD;
	IN7 : DWORD;
	IN8 : DWORD;
END_VAR
VAR_OUTPUT
	OUT1 : DWORD;
	OUT2 : DWORD;
	OUT3 : DWORD;
	OUT4 : DWORD;
	OUT5 : DWORD;
	OUT6 : DWORD;
	OUT7 : DWORD;
	OUT8 : DWORD;
	ID : BYTE;
END_VAR
VAR
	init : BOOL;
	i : INT;
	i2 : INT;
	index : INT;
	index2 : INT;
	ra : ARRAY[1..8] OF DWORD;
END_VAR

(*
version 1.0		15. may. 2011
programmer		ks
tested by			ks

NET_VAR_DWORD8 überträgt bidirektional acht DWORD vom Master zum Client
*)

IF NOT init THEN
	init := TRUE;
	X.ID_MAX := X.ID_MAX + USINT#1;
	ID := USINT_TO_BYTE(X.ID_MAX);
END_IF;

IF X.STATE > BYTE#0 AND X.ERROR_ID = BYTE#0 THEN
	index := X.index; (* PCWORX Workaround *)
	IF INT_TO_UINT(index + 34) > X.BUF_SIZE THEN  (* ID (1) + TYPE (1) + 8 x DWORD (4) *)
		X.ERROR_ID := ID;
	ELSE
		IF X.STATE = BYTE#1 THEN (* Daten schreiben *)
			ra[1] := IN1;
			ra[2] := IN2;
			ra[3] := IN3;
			ra[4] := IN4;
			ra[5] := IN5;
			ra[6] := IN6;
			ra[7] := IN7;
			ra[8] := IN8;
			X.S_BUF.BUFFER[index] := ID; (* ID *)
			index := index + 1;
			X.S_BUF.BUFFER[index] := BYTE#13; (* TYPE DWORD8 *)
			index := index + 1;
			FOR i2 := 1 TO 8 DO;
				FOR i := 1 TO 4 DO;
					X.S_BUF.BUFFER[index] := DWORD_TO_BYTE(ra[i2]);
					ra[i2] := ROR(ra[i2],8);
					index := index + 1;
				END_FOR;
			END_FOR;

		ELSIF X.STATE = BYTE#2 THEN (* Daten lesen *)
			index2 := index + 1; (* PCWORX Workaround *)
			IF X.R_BUF.BUFFER[index] <> ID OR X.R_BUF.BUFFER[index2] <> BYTE#13 THEN (* TYPE DWORD8 *)
				X.ERROR_ID := ID;
			ELSE
				index := index + 2;
				FOR i2 := 1 TO 8 DO;
					ra[i2] := DWORD#0;
					FOR i := 1 TO 4 DO;
						ra[i2] := ra[i2] OR BYTE_TO_DWORD(X.R_BUF.BUFFER[index]);
						ra[i2] := ROR(ra[i2],8);
						index := index + 1;
					END_FOR;
				END_FOR;
				OUT1 := ra[1];
				OUT2 := ra[2];
				OUT3 := ra[3];
				OUT4 := ra[4];
				OUT5 := ra[5];
				OUT6 := ra[6];
				OUT7 := ra[7];
				OUT8 := ra[8];
			END_IF;
		END_IF;
		X.index := index;
	END_IF;
END_IF;

(* revision history
ks	15.may. 2011	rev 1.0
	original version

*)

END_FUNCTION_BLOCK

// POUs/DEMO/Need Fixing/IRTRANS_DEMO
PROGRAM IRTRANS_DEMO
VAR
	IP_C : IP_C;
	S_BUF : NETWORK_BUFFER_SHORT;
	R_BUF : NETWORK_BUFFER_SHORT;
	IP_CONTROL2 : IP_CONTROL2;
	IRTRANS_DECODE : IRTRANS_DECODE;
	IRTRANS_RCV_4 : IRTRANS_RCV_4;
	DRIVER_4 : DRIVER_4;
	IRTRANS_SERVER : IRTRANS_SERVER;
	IRTRANS_SND_8_1 : IRTRANS_SND_8;
	IRTRANS_SND_8_2 : IRTRANS_SND_8;
	Q0: BOOL;
	Q1: BOOL;
	Q2: BOOL;
	Q3: BOOL;
	error: BOOL;
	error_server: DWORD;
	Send_1_0: BOOL := TRUE;
	Send_1_1: BOOL;
	Send_1_2: BOOL;
	Send_1_3: BOOL;
	Send_1_4: BOOL;
	Send_1_5: BOOL;
	Send_1_6: BOOL;
	Send_1_7: BOOL;
	Send_2_0: BOOL := TRUE;
	Send_2_1: BOOL;
	Send_2_2: BOOL;
	Send_2_3: BOOL;
	Send_2_4: BOOL;
	Send_2_5: BOOL;
	Send_2_6: BOOL;
	Send_2_7: BOOL;
	R_ENABLE: BOOL;
	S_ENABLE: BOOL;
	MODE: BOOL := FALSE;
	KEY_1: BYTE;
	KEY_2: BYTE;
END_VAR

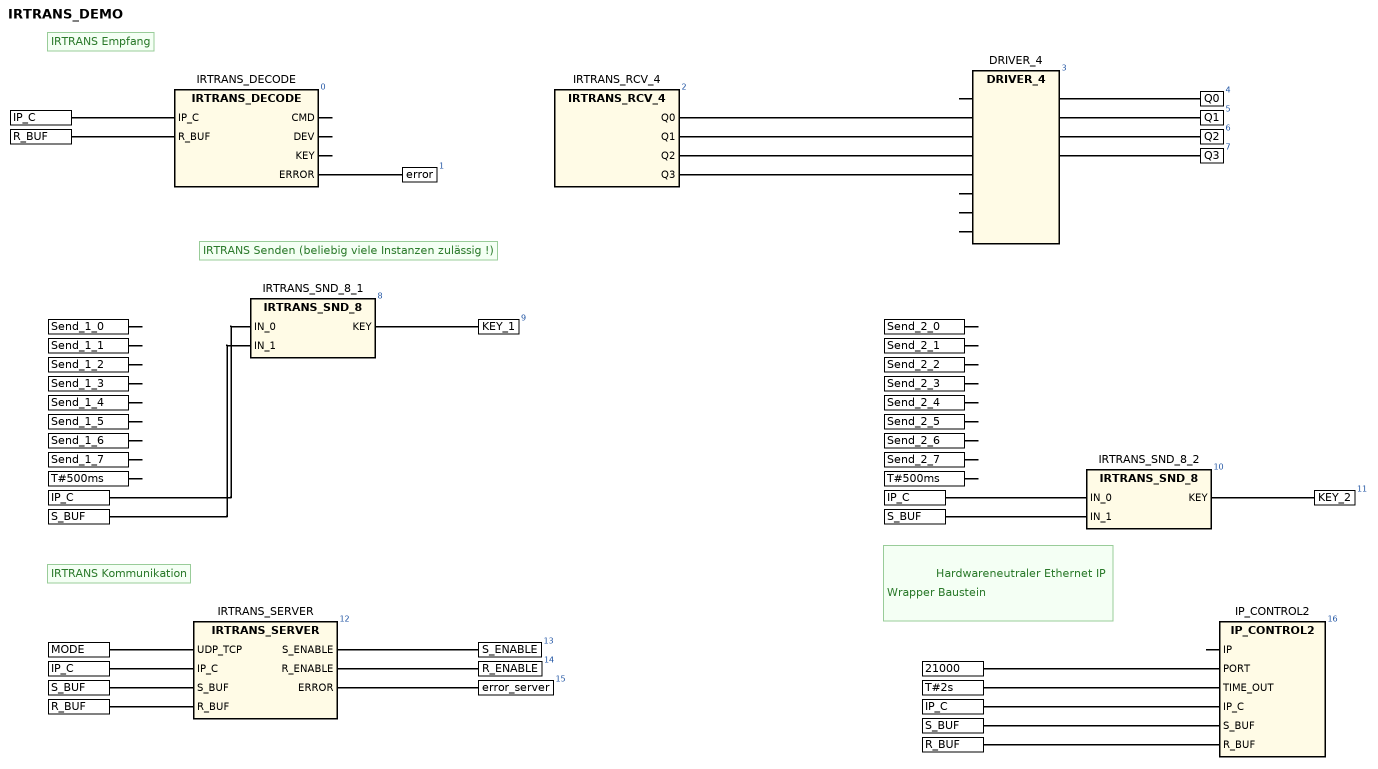
// note: 21 stored wires end on pins the file does not list and are not shown
// IRTRANS Empfang
IRTRANS_DECODE(IP_C := IP_C, R_BUF := R_BUF);
error := IRTRANS_DECODE.ERROR;
IRTRANS_RCV_4();
DRIVER_4(
    _in2 := IRTRANS_RCV_4.Q0,
    _in3 := IRTRANS_RCV_4.Q1,
    _in4 := IRTRANS_RCV_4.Q2,
    _in5 := IRTRANS_RCV_4.Q3);
Q0 := DRIVER_4._out1;
Q1 := DRIVER_4._out2;
Q2 := DRIVER_4._out3;
Q3 := DRIVER_4._out4;
// IRTRANS Senden (beliebig viele Instanzen zulässig !)
IRTRANS_SND_8_1(IN_0 := IP_C, IN_1 := S_BUF); // IRTRANS_SND_8
KEY_1 := IRTRANS_SND_8_1.KEY;
IRTRANS_SND_8_2(IN_0 := IP_C, IN_1 := S_BUF); // IRTRANS_SND_8
KEY_2 := IRTRANS_SND_8_2.KEY;
// IRTRANS Kommunikation
IRTRANS_SERVER(UDP_TCP := MODE, IP_C := IP_C, S_BUF := S_BUF, R_BUF := R_BUF);
S_ENABLE := IRTRANS_SERVER.S_ENABLE;
R_ENABLE := IRTRANS_SERVER.R_ENABLE;
error_server := IRTRANS_SERVER.ERROR;
// 							Hardwareneutraler Ethernet IP
// Wrapper Baustein
//
IP_CONTROL2(PORT := 21000, TIME_OUT := T#2s, IP_C := IP_C, S_BUF := S_BUF, R_BUF := R_BUF);
// Send_1_0: input not connected
// Send_1_1: input not connected
// Send_1_2: input not connected
// Send_1_3: input not connected
// Send_1_4: input not connected
// Send_1_5: input not connected
// Send_1_6: input not connected
// Send_1_7: input not connected
// Send_2_0: input not connected
// Send_2_1: input not connected
// Send_2_2: input not connected
// Send_2_3: input not connected
// Send_2_4: input not connected
// Send_2_5: input not connected
// Send_2_6: input not connected
// Send_2_7: input not connected
// T#500ms: input not connected
// T#500ms: input not connected

END_PROGRAM

// POUs/_HARDWARE/IP_CONTROL2
FUNCTION_BLOCK IP_CONTROL2
VAR_IN_OUT
	IP_C : IP_C; (* IP_Control Verwaltungsstruktur *)
	S_BUF : NETWORK_BUFFER_SHORT; (* Externer Sendbuffer *)
	R_BUF : NETWORK_BUFFER_SHORT; (* Externer Receivebuffer *)
END_VAR
VAR_INPUT
	IP : DWORD; (* IP Adresse *)
	PORT : WORD; (* Port Nummer *)
	TIME_OUT : TIME; (* Ueberwachungszeit Connect / Send / Receive *)
END_VAR
VAR
	c_time : UDINT; (* CONNECT-Time (Zeit bei nicht vorhandener Verbindung) *)
	s_time : UDINT; (* SEND-Time    (Zeit seit letzten Datensenden) *)
	r_time : UDINT; (* RECEIVE-Time (Zeit seit letztem Datenempfang) *)

	c_enable : BOOL; (* Connect: freigabe *)
	c_ip : DWORD; (* Connect: aktuelle IP-Adresse *)
	c_port : WORD; (* Connect: aktuelle Port-Nummer *)
	c_mode : BYTE; (* Connect: aktueller Mode UDP/TCP...... *)
	c_status : BYTE; (* Connect: Status (Errorcode) *)
	c_ready : BOOL; (* Connect: Verbindung aufgebaut *)
	c_ready_old : BOOL; (* Connect: letzter Zustand von c_ready für Flankenauswertung *)
	c_select : BOOL; (* non blocking mode - abfrage über select durchführen *)
	c_fdWrite : SOCKET_FD_SET;
	c_Timeout : SOCKET_TIMEVAL;

	s_total : INT; (* Send: Gesamtanzahl Bytes zum senden *)
	s_cur_pos : INT; (* Send: aktuelle Sendeposition *)
	s_cur_size : INT; (* Send: aktuelle Sendegroesse *)
	s_max_size : INT; (* Send: maximale Telegrammlänge fuer Senden *)
	s_start : BOOL; (* Send: Sende modus aktivieren *)
	s_active : BOOL; (* Send: Daten senden ist aktiv *)
	s_req : BOOL; (* Send: Start Daten senden *)
	s_done : BOOL; (* Send: ohne Fehler beendet *)
	s_status : BYTE; (* Send: Status (Errorcodes) *)

	r_status : BYTE; (* Receive: Status (Errorcodes) *)
	r_count : INT; (* Receive: Anzahl empfangener Bytes *)
	r_offset : INT; (* Receive: aktuelle Position in externen Receivebuffer *)
	r_max_size : INT; (* Receive: groesse des externen Empfangbuffers*)

	new_connection : BOOL; (* Neue Verbindungsparameter vorhanden *)
	tx : DWORD; (* letzter zeitwert *)
	error_time : DWORD; (* aktueller Timeout-Wert *)

	state: BYTE; (* schrittmerker für connect *)
	server_socket : RTS_IEC_HANDLE:= RTS_INVALID_HANDLE;                // Handle Pointing to our Socket
	socket : RTS_IEC_HANDLE:= RTS_INVALID_HANDLE;
	//server_socket : DINT:= RTS_INVALID_HANDLE;
	//socket : DINT:= RTS_INVALID_HANDLE;
	sockaddr : SOCKADDRESS;
	sockaddr_size : DWORD;
	plc_841 : BOOL;
	plc_881 : BOOL;
	dint_true : DINT := 1;
	bytes_received : DINT;
	bytes_sent : DINT;
	udp_mode : BOOL;

	pResult : UDINT; //Needed for V3 Lib
	FunctionResult 	: UDINT ;   
  	tAddress                	: INADDR;                           // Strucutre to define our internet address
	TESTtAddress               	: INADDR;   
	(*LOG_MSG : LOG_MSG;
	_debug_enable : BOOL := TRUE;
	debug_index : INT;
	debug_ID : INT;
	debug_lasterror : DWORD;
	debug_last_id : INT := 255;
	state_last: BYTE;*)

END_VAR

VAR CONSTANT
	STOP : BYTE := 0;
	TS_INIT: BYTE := 1;
	TS_OPEN : BYTE:= 2;

	UDP_INIT : BYTE:= 31;

	TC_INIT : BYTE:= 51;
	TC_CONNECT : BYTE:= 52;

	C_WAIT : BYTE:= 250;
	C_CLOSE : BYTE:= 251;

END_VAR

(*

version 1.9		26. Feb. 2012
programmer 		ks
tested by			ks

IP_CONTROL ist ein Wrapper-Baustein um eine Hersteller neutrale Schnittstelle zum Ethernet zu schaffen
*)

(* ---------------------- Debug-Message ----------------------------*)
(*IF _debug_enable THEN
	IF IP_C.FIFO.ID > BYTE#0 THEN (* nur wenn Teilnehmer ID's vorhanden sind *)
		debug_index := IP_C.FIFO.NR;
		debug_ID := BYTE_TO_INT(IP_C.FIFO.X[debug_index]);
	END_IF;
END_IF;*)
(* -----------------------------------------------------------------------------*)

(* read system time *)
tx := T_PLC_MS();

IF IP_C.C_PORT = 0 THEN
	IP_C.C_PORT := PORT; (* uebergebenen PORT durch parametrierten PORT ersetzen *)
END_IF;
IF IP_C.C_IP = 0 AND IP_C.C_MODE < 4 THEN
	IP_C.C_IP := IP; (* uebergebene IP durch paramtrierte IP ersetzen *)
END_IF;

new_connection := c_ip <> IP_C.C_IP OR c_mode <> IP_C.C_MODE OR c_port <> IP_C.C_PORT; (* neue Verbindungs erwünscht ? *)
c_enable := IP_C.C_ENABLE AND NOT new_connection;

IF IP_C.C_ENABLE AND IP_C.ERROR = 0 AND state = STOP THEN (* Freigabe,kein Fehler,kein Socket offen *)
	c_ip   := IP_C.C_IP;
	c_mode := IP_C.C_MODE;
	c_port := IP_C.C_PORT;
	plc_841 := ADR(%MW0)=16#30000000; (*750-841*)
	plc_881 := ADR(%MW0)=16#20000000; (*750-881*)
	udp_mode := C_MODE.0; (* Mode 1,3,5 = udp *)

	error_time := TIME_TO_DWORD(MAX(T#200ms,TIME_OUT));
	IP_C.TIME_RESET := TRUE; (* Alle Timer ruecksetzen *)

	r_max_size := UINT_TO_INT(SIZEOF(R_BUF.BUFFER));
	s_max_size := UINT_TO_INT(SIZEOF(S_BUF.BUFFER));

	IF C_MODE.0 THEN (* Mode: 1,3,5 = UDP CLIENT/SERVER *)
		state := UDP_INIT;
	ELSIF C_MODE = 0 THEN (* Mode: 0 = TCP CLIENT *)
		state := TC_INIT;
	ELSE
		state := TS_INIT; (* Mode: 2,4 = TCP SERVER *)
	END_IF;

	(* ---------------------- Debug-Message ----------------------------*)
	(*IF _debug_enable THEN
		LOG_CL.NEW_MSG := 'IP_CON: MODE ~1 / IP ~2 / PORT ~3 /ID ~6';
		LOG_CL.PRINTF[1] := BYTE_TO_STRING(C_MODE);
		LOG_CL.PRINTF[2] := IP4_TO_STRING(c_ip);
		LOG_CL.PRINTF[3] := WORD_TO_STRING(c_port);
		LOG_CL.PRINTF[6] := INT_TO_STRING(debug_ID);
		LOG_MSG();
	END_IF;*)
	(* -----------------------------------------------------------------------------*)

END_IF;

(* ---------------------- Debug-Message ----------------------------*)
(*IF  _debug_enable THEN
	IF state <> state_last THEN
		LOG_CL.NEW_MSG := 'IP_STEP ~1 -IP_ID ~6';
		LOG_CL.PRINTF[1] := BYTE_TO_STRING(state);
		LOG_CL.PRINTF[6] := INT_TO_STRING(debug_ID);
		LOG_MSG();
		state_last := state;
	END_IF;
END_IF;*)
(* -----------------------------------------------------------------------------*)

IF IP_C.TIME_RESET THEN (* Alle Timer ruecksetzen *)
	IP_C.TIME_RESET := FALSE; (* Reset rücksetzen *)
	c_time := tx; (* Connect Timer ruecksetzen *)
	s_time := tx; (* Send Timer ruecksetzen *)
	r_time := tx; (* Receive Timer ruecksetzen *)

	c_status := BYTE#0; (* letzten Connect Fehler rücksetzen *)
	s_status := BYTE#0; (* letzten Send Fehler rücksetzen *)
	r_status := BYTE#0; (* letzten Receive Fehler rücksetzen *)
END_IF;

(* ---------------------------------------------- *)

CASE state OF

UDP_INIT: (* UDP_CLIENT + SERVER *)
	socket := SysSockCreate(SOCKET_AF_INET, SOCKET_DGRAM, SOCKET_IPPROTO_IP, ADR(pResult));
	IF socket < 0 THEN
		c_status := 1; (* SysSockCreate failed *)
		state := C_CLOSE;
	ELSE
		FunctionResult :=SysSockSetOption(socket, SOCKET_SOL, SOCKET_SO_BROADCAST, ADR(dint_true), SIZEOF(dint_true)); (* allow broadcast *)
		FunctionResult :=SysSockIoctl(socket, SOCKET_FIONBIO, ADR(dint_true)); (* put socket in non-blocking mode *)
		sockaddr.sin_family := SOCKET_AF_INET;
		sockaddr.sin_port := SysSockHtons(c_port);
		sockaddr.sin_addr.ulAddr := SEL(c_mode = 1, SOCKET_INADDR_ANY, SysSockNtohl(c_ip));

		IF c_mode >= 2 THEN (* SERVER Mode *)
			FunctionResult := SysSockBind(socket, ADR(sockaddr), SIZEOF(sockaddr));
			IF FunctionResult=0 THEN
				c_ready := TRUE; (* Connected *)
				state:= C_WAIT;
			ELSE
				c_status := 2; (* SysSockBind failed *)
				state := C_CLOSE;
			END_IF;
		ELSE
			c_ready := TRUE; (* Connected *)
			state:= C_WAIT;
		END_IF;
	END_IF;

(* ---------------------------------------------- *)

TC_INIT: (* TCP-CLIENT (AKTIV) *)
	// Create handle to ethernet socket to send messages
	socket        := SysSockCreate(SOCKET_AF_INET, SOCKET_STREAM, SOCKET_IPPROTO_TCP, ADR(pResult)); 	
	IF socket < 0 THEN
		c_status := 1;  (* SysSockCreate failed *)
		state := C_CLOSE;
	ELSE
		IF plc_841 OR plc_881 THEN
			FunctionResult :=SysSockSetOption(socket,6,SOCKET_TCP_NODELAY, ADR(dint_true), SIZEOF(dint_true)); (* Set Push-Bit *)
		END_IF;
		// Set option for local address reuse
		FunctionResult :=SysSockSetOption(socket, SOCKET_SOL, SOCKET_SO_REUSEADDR, ADR(dint_true), SIZEOF(dint_true));
		// Set option for keepalive
		//FunctionResult := SysSockSetOption(socket, SOCKET_SOL, SOCKET_SO_KEEPALIVE, ADR(dint_true), SIZEOF(dint_true));
		
        //Moved to After Connect 
		//FunctionResult :=SysSockIoctl(socket, SOCKET_FIONBIO, ADR(dint_true)); (* NonBlocking mode *)
		
		sockaddr.sin_family := SOCKET_AF_INET;
		sockaddr.sin_port := SysSockNtohs(c_port);
		sockaddr.sin_addr.ulAddr  := SysSockNtohl(c_ip);
		c_select := FALSE;
		state := TC_CONNECT;
	END_IF;

(* ---------------------------------------------- *)

TC_CONNECT:
	IF NOT c_enable OR c_status = 255 THEN (* keine freigabe oder connect timeout *)
			state:= C_CLOSE;
	ELSE
		IF c_select = FALSE THEN
			FunctionResult:=SysSockConnect(socket,ADR(sockaddr),SIZEOF(sockaddr));
			IF FunctionResult=0 THEN
				FunctionResult :=SysSockIoctl(socket, SOCKET_FIONBIO, ADR(dint_true)); (* NonBlocking mode *)
				c_ready := TRUE; (* Connected *)
				state:= C_WAIT;
			ELSE
				(* Connect durchgeführt, aber noch nicht verbunden, dann optional mit select-abfrage weitermachen *)
				c_select := SYSLIBSOCKETS_OPTION.0; (* Bit 0 = TCP-Client - use SysSockselect *)
			END_IF;
		ELSE
			c_Timeout.tv_sec := 0;
			c_Timeout.tv_usec := 0;
			c_fdWrite.fd_count := 1;
			c_fdWrite.fd_array[0] := socket;
			IF SysSockSelect(SOCKET_FD_SETSIZE,0,ADR(c_fdWrite),0, ADR(c_Timeout), ADR(pResult)) > 0 THEN
				c_ready := TRUE; (* Connected *)
				state:= C_WAIT;
			END_IF;
		END_IF;
	END_IF;

(* ---------------------------------------------- *)

TS_INIT: (* TCP-SERVER (PASSIV) *)
	server_socket := SysSockCreate(SOCKET_AF_INET, SOCKET_STREAM, SOCKET_IPPROTO_IP, ADR(pResult)); (* Create Socket *)
	IF server_socket = RTS_INVALID_HANDLE THEN
		c_status := 1; (* SysSockCreate failed *)
		state:= C_CLOSE;
	ELSE (* Address bindings *)
		SysSockSetOption( server_socket, SOCKET_SOL, SOCKET_SO_REUSEADDR, ADR(dint_true), SIZEOF(dint_true) );
		sockaddr.sin_family:= SOCKET_AF_INET;
		sockaddr.sin_port := SysSockHtons(c_port);
		sockaddr.sin_addr.ulAddr  := SOCKET_INADDR_ANY;
		IF NOT SysSockBind(server_socket, ADR(sockaddr), SIZEOF(sockaddr)) = 0 THEN
			c_status := 2; (* SysSockBind failed *)
			state := C_CLOSE;
		ELSIF NOT SysSockListen(server_socket, 1) = 0 THEN (* erzeugt Warteschlange für eine Verbindung *)
			c_status := 3; (* SysSockListen failed *)
			state:= C_CLOSE;
		ELSE
			SysSockIoctl(server_socket, SOCKET_FIONBIO, ADR(dint_true)); (* NonBlocking mode *)
			state:= TS_OPEN;
		END_IF;
	END_IF;

(* ---------------------------------------------- *)

TS_OPEN: (* Waiting for incomming connection *)
	sockaddr_size := SIZEOF(sockaddr);
	socket := SysSockAccept(server_socket, ADR(sockaddr), ADR(sockaddr_size), ADR(pResult));

	IF socket <> RTS_INVALID_HANDLE THEN (* neuer Verbindungswunsch vorhanden *)
		IF c_mode = BYTE#2 AND sockaddr.sin_addr.ulAddr <> SysSockNtohl(c_ip) THEN (* Mode 2 = TCP + PASSIVE + PORT + IP  auf richtige Partner-IP prüfen *)
			state:= C_CLOSE;
		ELSE
			IF plc_841 OR plc_881 THEN
				SysSockSetOption(socket, 6, SOCKET_TCP_NODELAY, ADR(dint_true), SIZEOF(dint_true)); (* Set Push-Bit *)
			END_IF;
			SysSockIoctl(socket, SOCKET_FIONBIO, ADR(dint_true)); (* NonBlocking mode *)
			c_ready := TRUE; (* Connected *)
			state := C_WAIT;
		END_IF;
	ELSIF NOT c_enable THEN (* keine freigabe mehr ? *)
			state:= C_CLOSE;
	END_IF;

(* ---------------------------------------------- *)

C_WAIT: (* Warten auf Anforderung für Beenden *)
	IF NOT c_enable OR NOT c_ready THEN
		state:= C_CLOSE;
	END_IF

(* ---------------------------------------------- *)

C_CLOSE: (* Close the Sockets *)
	c_ready := FALSE;
	IF socket >= 0 THEN
		IF (NOT plc_841) AND (NOT plc_881) THEN
			SysSockShutdown(socket, 0); (* 870 *)
		END_IF;
		SysSockClose(socket);
		socket := RTS_INVALID_HANDLE;
	END_IF
	IF server_socket >= 0 THEN
		IF (NOT plc_841) AND (NOT plc_881) THEN
			SysSockShutdown(server_socket, 0); (* 870 *)
		END_IF;
		SysSockClose(server_socket);
		server_socket := RTS_INVALID_HANDLE;
	END_IF
	state:= STOP;
END_CASE;

(* ---------------------------------------------- *)

IF c_ready THEN
	IF NOT c_ready_old THEN (* Verbindung aufgebaut - positive Flanke erkannt *)
		IP_C.C_STATE := 254;
		IP_C.TIME_RESET := TRUE; (* Alle Timer ruecksetzen *)
		(* ---------------------- Debug-Message ----------------------------*)
		(*IF _debug_enable THEN
			LOG_CL.NEW_MSG := 'IP_CON: CONNECTED -IP_ID ~6';
			LOG_CL.PRINTF[6] := INT_TO_STRING(debug_ID);
			LOG_MSG();
		END_IF;*)
		(* -----------------------------------------------------------------------------*)
	ELSE
		IP_C.C_STATE := 255; (* Verbindung ist aufgebaut *)
	END_IF;
ELSE
	IF c_ready_old THEN (* Verbindung abgebaut - negative Flanke erkannt *)
		IP_C.C_STATE := 1;
		IP_C.MAILBOX[1] := 0; (* Receive Info rücksetzen *)
		IP_C.MAILBOX[2] := 0; (* Send-Pause rücksetzen *)
		IP_C.MAILBOX[3] := 0; (* Receive-Pause rücksetzen *)
		IF NOT new_connection THEN
			s_active := FALSE; (* Sendeaktivitäten stoppen *)
			s_req := FALSE; (* Sendefreigabe rücksetzen *)
			S_BUF.SIZE := 0; (* Sendelänge löschen *)
			(*IP_C.TIME_RESET := TRUE;*) (* Alle Timer ruecksetzen *)
		END_IF;
		(* ---------------------- Debug-Message ----------------------------*)
		(*IF _debug_enable THEN
			LOG_CL.NEW_MSG := 'IP_CON: DISCONNECTED';
			LOG_MSG();
		END_IF;*)
		(* -----------------------------------------------------------------------------*)
	ELSE
		IP_C.C_STATE := 0; (* Verbindung ist abgebaut *)
	END_IF;
END_IF;

c_ready_old := c_ready;

(* Der Datenempfang wird angehalten solange ein Sendevorgang läuft *)
(* sonst kann es vorkommen das die Antwort-daten schon empfangen werden, *)
(* bevor der Sendevorgang vom programm abgeschlossen wurde *)

IF c_ready AND NOT s_active AND IP_C.MAILBOX[3] = 0 THEN
	IF R_BUF.SIZE >= INT_TO_UINT(r_max_size) THEN
		R_BUF.SIZE := UINT#0;
		r_status := 254; (* Empfangsbuffer wegen Überlauf rückgesetzt *)
	END_IF;

	r_offset := SEL(udp_mode,UINT_TO_INT(R_BUF.SIZE),0);
	r_count := r_max_size - r_offset;

	IF udp_mode THEN
		bytes_received := SysSockRecvFrom(socket, ADR(R_BUF.BUFFER), r_count, 0, ADR(sockaddr), SIZEOF(sockaddr), ADR(pResult));

		IF c_mode = BYTE#3 AND sockaddr.sin_addr.ulAddr <> SysSockNtohl(c_ip) THEN (* Mode 3 = UDP + PASSIVE + PORT + IP  auf richtige Partner-IP prüfen *)
			bytes_received := 0;
			R_BUF.SIZE := UINT#0;
			sockaddr.sin_port := SysSockNtohs(c_port);
			sockaddr.sin_addr.ulAddr  := SysSockNtohl(c_ip);
		END_IF;

	ELSE
		bytes_received := SysSockRecv(socket, ADR(R_BUF.BUFFER[r_offset]), r_count, 0, ADR(pResult));
	END_IF;

	CASE pResult OF  //Added for Version3 Libs
		518:  bytes_received:=-1; //Connection OKAY just no data and do not want to BIND
		521:  bytes_received:=0; //Connection has been refused by the remote host 
		523:  bytes_received:=0; //The host has not been found  
		524:  bytes_received:=0; //Host is unreachable  
		526:  bytes_received:=0; //The socket is not connected  
		527:  bytes_received:=0; //Shutdown has been called on the socket  
		529:  bytes_received:=0; //Socket has been gracefully closed. No more send/receives allowed	 
	END_CASE

	
	(*UDP: IPC returns -1 if no data available or error occured,841 returns -1 if error occured and 0 if no data available*)
	CASE bytes_received OF
	-2147483648..-1: ; (* No data available or error occured *)
	 0: IF NOT udp_mode OR pResult<>518 THEN (* TCP-Mode: socket wurde von remote geschlossen *)
			c_status := 253;
			c_ready := FALSE;
		END_IF;
	ELSE (* daten wurden empfangen *)
  		r_time := tx; (* Receive Timer ruecksetzen *)
		R_BUF.SIZE := INT_TO_UINT(r_offset) + DINT_TO_UINT(bytes_received); (* aktuelle buffersize eintragen *)
		IP_C.MAILBOX[1] := IP_C.MAILBOX[1] + 1; (* Receive Info *)
		IF IP_C.MAILBOX[1] = 0 THEN IP_C.MAILBOX[1] := 1; END_IF;

		(* ---------------------- Debug-Message ----------------------------*)
		(*IF _debug_enable THEN
			LOG_CL.NEW_MSG := 'IP_REC DATA: POS: ~1 : SIZE: ~2 TOTAL ~3 -IP_ID ~6';
			LOG_CL.PRINTF[1] := INT_TO_STRING(r_offset);
			LOG_CL.PRINTF[2] := INT_TO_STRING(r_count);
			LOG_CL.PRINTF[3] := UINT_TO_STRING(R_BUF.SIZE);
			LOG_CL.PRINTF[6] := INT_TO_STRING(debug_ID);
			LOG_MSG();
		END_IF;*)
		(* -----------------------------------------------------------------------------*)

	END_CASE
END_IF;

(* ---------------------------------------------- *)

IF S_BUF.SIZE > 0 THEN
	IF c_ready AND c_enable THEN
		IF NOT s_active AND IP_C.MAILBOX[2] = 0 THEN
			(* Gesamtanzahl an Bytes limitieren und uebergeben *)
			s_total := LIMIT(0,UINT_TO_INT(S_BUF.SIZE),r_max_size);
			s_cur_pos  := 0;
			s_cur_size := 0;
			s_start := TRUE; (* Daten kopieren und senden anstossen *)
			s_active := TRUE; (* Sende-Betrieb aktivieren *)
			(* ---------------------- Debug-Message ----------------------------*)
			(*IF _debug_enable THEN
				LOG_CL.NEW_MSG := 'IP_SEN INIT: TOTAL: ~1 -IP_ID ~6';
				LOG_CL.PRINTF[1] := INT_TO_STRING(S_TOTAL);
				LOG_CL.PRINTF[6] := INT_TO_STRING(debug_ID);
				LOG_MSG();
			END_IF;*)
			(* -----------------------------------------------------------------------------*)
		END_IF;

		IF s_done OR s_start THEN (* Daten senden aktiv *)

			s_start := FALSE;
			s_cur_pos := s_cur_pos + s_cur_size; (* neue Sende-Datenposition bestimmen *)
			IF s_total > s_cur_pos THEN (* weitere Daten zum senden vorhanden ? *)
				s_cur_size := s_total - s_cur_pos;
				s_cur_size := LIMIT(0, s_cur_size, s_max_size); (* Telegrammlänge begrenzen *)
				(* ---------------------- Debug-Message ----------------------------*)
				(*IF _debug_enable THEN
					LOG_CL.NEW_MSG := 'IP_SEN DATA: POS: ~1 : SIZE: ~2 TOTAL ~3 -IP_ID ~6';
					LOG_CL.PRINTF[1] := INT_TO_STRING(S_CUR_POS);
					LOG_CL.PRINTF[2] := INT_TO_STRING(S_CUR_SIZE);
					LOG_CL.PRINTF[3] := INT_TO_STRING(S_TOTAL);
					LOG_CL.PRINTF[6] := INT_TO_STRING(debug_ID);
					LOG_MSG();
				END_IF;*)
				(* -----------------------------------------------------------------------------*)
				s_time := tx; (* Send Timer ruecksetzen *)
				r_time := tx; (* Receive Timer ruecksetzen *)
				s_req := TRUE;

			ELSE
				(* keine weitere Sendedaten vorhanden -> Senden beenden *)
				s_req := FALSE;
				s_active := FALSE;
				S_BUF.SIZE := 0;
				(* ---------------------- Debug-Message ----------------------------*)
				(*IF _debug_enable THEN
					LOG_CL.NEW_MSG := 'IP_SEN FINISH -IP_ID ~6';
					LOG_CL.PRINTF[6] := INT_TO_STRING(debug_ID);
					LOG_MSG();
				END_IF;*)
				(* -----------------------------------------------------------------------------*)
			END_IF;
		END_IF;
	END_IF;
END_IF;

IF s_req THEN
	s_done := FALSE;
	IF udp_mode THEN
		bytes_sent := SysSockSendTo(socket, ADR(S_BUF.BUFFER[s_cur_pos]), s_cur_size, 0, ADR(sockaddr), SIZEOF(sockaddr), ADR(pResult));
	ELSE
		bytes_sent := SysSockSend(socket, ADR(S_BUF.BUFFER[s_cur_pos]), s_cur_size, 0, ADR(pResult));
	END_IF;

	CASE bytes_sent OF
	-2147483648..-1:	; (* ERROR: Noch nicht bereit um Daten aufzunehmen -> nächsten Zyklus wieder probieren *)
	 0: IF NOT udp_mode THEN (* TCP-Mode: socket wurde von remote geschlossen *)
			c_status := 253;
			c_ready := FALSE;
		END_IF;
	ELSE
		s_done := TRUE;
		s_cur_size := DINT_TO_INT(bytes_sent); (* Anzahl der wirklich versendeten Bytes übernehmen *)
		(* ---------------------- Debug-Message ----------------------------*)
		(*IF _debug_enable THEN
			LOG_CL.NEW_MSG := 'IP_SEN SEND_COUNT ~1 -IP_ID ~6';
			LOG_CL.PRINTF[1] := DINT_TO_STRING(s_cur_size);
			LOG_CL.PRINTF[6] := INT_TO_STRING(debug_ID);
			LOG_MSG();
		END_IF;*)
		(* -----------------------------------------------------------------------------*)
	END_CASE
END_IF;

(* ---------------------------------------------- *)

IF IP_C.R_OBSERVE = FALSE OR s_active THEN
    r_time := tx;
END_IF;

IF c_status = 0 AND tx - c_time > error_time AND c_enable AND NOT c_ready AND c_mode < 2 THEN (* Connect Timeout *)
	c_status := 255; (* Timeout-Fehler ausgeben *)
END_IF;
IF s_status = 0 AND tx - s_time > error_time AND s_active THEN (* Send Timeout *)
	s_status := 255; (* Timeout-Fehler ausgeben *)
END_IF;
IF r_status = 0 AND tx - r_time > error_time AND c_ready AND IP_C.R_OBSERVE THEN (* Receive Timeout *)
	r_status := 255; (* Timeout-Fehler ausgeben *)
END_IF;

IP_C.ERROR := DWORD_OF_BYTE(c_status,s_status,r_status,0);

(* ---------------------- Debug-Message ----------------------------*)
(*IF  _debug_enable THEN
	IF (IP_C.ERROR <> debug_lasterror) THEN
		LOG_CL.NEW_MSG := 'IP_ERROR ~1 -IP_ID ~6';
		LOG_CL.PRINTF[1] := DWORD_TO_STRING(IP_C.ERROR);
		LOG_CL.PRINTF[6] := INT_TO_STRING(debug_ID);
		LOG_MSG();

		debug_lasterror := IP_C.ERROR;
		debug_last_id := debug_ID;
	END_IF;
END_IF;*)
(* -----------------------------------------------------------------------------*)

(* revision history
ks	18. oct. 2008	rev 1.0
	original version
ks	05. jan. 2009	rev 1.1
	zusätzlichen Parameter "Port" hinzugefügt, und Code bei Verbindungsaufbau angepasst
ks	28. feb. 2009	rev 1.2
	connect code angepasst und verkürzung der zyklen bei Send
ks	20. oct. 2009	rev 1.3
	network_buffer basis 0
ks	06. dec. 2009	rev 1.4
	receive_count MAILBOX[1]
ks	10. nov. 2010	rev 1.5
	send_pause MAILBOX[2] and receive_pause MAILBOX[3] 
ks	07. feb. 2011	rev 1.6
	Fehlercode 253 bei Remote-Verbindungsabbruch
ks	30. may. 2011	rev 1.7
	Fehler bei Empfangsüberwachung
ks	26. july. 2011	rev 1.8
	Error-Reset, diverse optimierungen 
ks	26. feb. 2012	rev 1.9
	Code-Optimierung für höhere kompatibilität

*)

END_FUNCTION_BLOCK

// POUs/NET_VAR/NET_VAR_REAL8
FUNCTION_BLOCK NET_VAR_REAL8
VAR_IN_OUT
	X : NET_VAR_DATA;
END_VAR
VAR_INPUT
	IN1 : REAL;
	IN2 : REAL;
	IN3 : REAL;
	IN4 : REAL;
	IN5 : REAL;
	IN6 : REAL;
	IN7 : REAL;
	IN8 : REAL;
END_VAR
VAR_OUTPUT
	OUT1 : REAL;
	OUT2 : REAL;
	OUT3 : REAL;
	OUT4 : REAL;
	OUT5 : REAL;
	OUT6 : REAL;
	OUT7 : REAL;
	OUT8 : REAL;
	ID : BYTE;
END_VAR
VAR
	init : BOOL;
	i : INT;
	i2 : INT;
	index : INT;
	index2 : INT;
	r_dw : DWORD;
	ra : ARRAY[1..8] OF REAL;
END_VAR

(*
version 1.0		15. may. 2011
programmer		ks
tested by			ks

NET_VAR_REAL8 überträgt bidirektional acht REAL-Werte vom Master zum Client
*)

IF NOT init THEN
	init := TRUE;
	X.ID_MAX := X.ID_MAX + USINT#1;
	ID := USINT_TO_BYTE(X.ID_MAX);
END_IF;

IF X.STATE > BYTE#0 AND X.ERROR_ID = BYTE#0 THEN
	index := X.index; (* PCWORX Workaround *)
	IF INT_TO_UINT(index + 34) > X.BUF_SIZE THEN (* ID (1) + TYPE (1) + 8 x REAL (4) *)
		X.ERROR_ID := ID;
	ELSE
		IF X.STATE = BYTE#1 THEN (* Daten schreiben *)
			ra[1] := IN1;
			ra[2] := IN2;
			ra[3] := IN3;
			ra[4] := IN4;
			ra[5] := IN5;
			ra[6] := IN6;
			ra[7] := IN7;
			ra[8] := IN8;
			X.S_BUF.BUFFER[index] := ID; (* ID *)
			index := index + 1;
			X.S_BUF.BUFFER[index] := BYTE#15; (* TYPE REAL8 *)
			index := index + 1;
			FOR i2 := 1 TO 8 DO;
				r_dw := OSCAT_BASIC.REAL_TO_DW(X:=ra[i2]);
				FOR i := 1 TO 4 DO;
					X.S_BUF.BUFFER[index] := DWORD_TO_BYTE(r_dw);
					r_dw := ROR(r_dw,8);
					index := index + 1;
				END_FOR;
			END_FOR;

		ELSIF X.STATE = BYTE#2 THEN (* Daten lesen *)
			index2 := index + 1; (* PCWORX Workaround *)
			IF X.R_BUF.BUFFER[index] <> ID OR X.R_BUF.BUFFER[index2] <> BYTE#15 THEN (* TYPE REAL8 *)
				X.ERROR_ID := ID;
			ELSE
				index := index + 2;
				FOR i2 := 1 TO 8 DO;
					r_dw := DWORD#0;
					FOR i := 1 TO 4 DO;
						r_dw := r_dw OR BYTE_TO_DWORD(X.R_BUF.BUFFER[index]);
						r_dw := ROR(r_dw,8);
						index := index + 1;
					END_FOR;
					ra[i2] := OSCAT_BASIC.DW_TO_REAL(X:=r_dw);
				END_FOR;
				OUT1 := ra[1];
				OUT2 := ra[2];
				OUT3 := ra[3];
				OUT4 := ra[4];
				OUT5 := ra[5];
				OUT6 := ra[6];
				OUT7 := ra[7];
				OUT8 := ra[8];
			END_IF;
		END_IF;
		X.index := index;
	END_IF;
END_IF;

(* revision history
ks	15.may. 2011	rev 1.0
	original version

*)

END_FUNCTION_BLOCK

// POUs/NET_VAR/NET_VAR_STRING
FUNCTION_BLOCK NET_VAR_STRING
VAR_IN_OUT
	IN : STRING(OSCAT_BASIC.STRING_LENGTH);
	OUT : STRING(OSCAT_BASIC.STRING_LENGTH);
	X : NET_VAR_DATA;
END_VAR
VAR_OUTPUT
	ID : BYTE;
END_VAR
VAR
	init : BOOL;
	len_str : INT;
	index : INT;
	index2 : INT;
END_VAR

(*
version 1.0		15. may. 2011
programmer		ks
tested by			ks

NET_VAR_STRING überträgt bidirektional einen STRING vom Master zum Client
*)

IF NOT init THEN
	init := TRUE;
	X.ID_MAX := X.ID_MAX + USINT#1;
	ID := USINT_TO_BYTE(X.ID_MAX);
END_IF;

IF X.STATE > BYTE#0 AND X.ERROR_ID = BYTE#0 THEN
	index := X.index; (* PCWORX Workaround *)
	IF X.STATE = BYTE#1 THEN (* Daten schreiben *)
		len_str := LEN(IN);
		IF INT_TO_UINT(index + 3 + len_str) > X.BUF_SIZE THEN
			X.ERROR_ID := ID;
		ELSE
			X.S_BUF.BUFFER[index] := ID; (* ID *)
			index := index + 1;
			X.S_BUF.BUFFER[index] := BYTE#6; (* TYPE REAL *)
			index := index + 1;
			X.S_BUF.BUFFER[index] := INT_TO_BYTE(len_str); (* Anzahl der Bytes *)
			index := index + 1;
			OSCAT_BASIC._STRING_TO_BUFFER(STR:=IN,POS:=index,PT:=ADR(X.S_BUF.BUFFER),SIZE:=X.BUF_SIZE);
			index := index + len_str;
		END_IF;
	ELSIF X.STATE = BYTE#2 THEN (* Daten lesen *)
		index2 := index + 1; (* PCWORX Workaround *)
		IF X.R_BUF.BUFFER[index] <> ID OR X.R_BUF.BUFFER[index2] <> BYTE#6 THEN
			X.ERROR_ID := ID;
		ELSE
			index := index + 2;
			len_str := BYTE_TO_INT(X.R_BUF.BUFFER[index]);
			index2 := index + 1;
			index := index2 + len_str;
			IF len_STR > 0 THEN
				OUT := OSCAT_BASIC.BUFFER_TO_STRING(PT:=ADR(X.R_BUF.BUFFER),SIZE:=X.BUF_SIZE,START:=INT_TO_UINT(index2),STOP:=INT_TO_UINT(index - 1));
			ELSE
				OUT := '';
			END_IF;
		END_IF;
	END_IF;
	X.index := index;
END_IF;

(* revision history
ks	15.may. 2011	rev 1.0
	original version

*)

END_FUNCTION_BLOCK

// POUs/NET_VAR/NET_VAR_X8
FUNCTION_BLOCK NET_VAR_X8
VAR_IN_OUT
	X : NET_VAR_DATA;
END_VAR
VAR_INPUT
	IN_REAL1 : REAL;
	IN_REAL2 : REAL;
	IN_DINT1 : DINT;
	IN_DINT2 : DINT;
	IN_UDINT1 : UDINT;
	IN_UDINT2 : UDINT;
	IN_DWORD1 : DWORD;
	IN_DWORD2 : DWORD;
END_VAR
VAR_OUTPUT
	OUT_REAL1 : REAL;
	OUT_REAL2: REAL;
	OUT_DINT1 : DINT;
	OUT_DINT2 : DINT;
	OUT_UDINT1 : UDINT;
	OUT_UDINT2 : UDINT;
	OUT_DWORD1 : DWORD;
	OUT_DWORD2 : DWORD;
	ID : BYTE;
END_VAR
VAR
	init : BOOL;
	i : INT;
	i2 : INT;
	index : INT;
	index2 : INT;
	ra : ARRAY[1..8] OF DWORD;
END_VAR

(*
version 1.0		15. may. 2011
programmer		ks
tested by			ks

NET_VAR_X8 überträgt bidirektional 2x REAL,2x DINT,2x UDINT,2x DWORD vom Master zum Client
*)

IF NOT init THEN
	init := TRUE;
	X.ID_MAX := X.ID_MAX + USINT#1;
	ID := USINT_TO_BYTE(X.ID_MAX);
END_IF;

IF X.STATE > BYTE#0 AND X.ERROR_ID = BYTE#0 THEN
	index := X.index; (* PCWORX Workaround *)
	IF INT_TO_UINT(index + 34) > X.BUF_SIZE THEN  (* ID (1) + TYPE (1) + 8 x DWORD (4) *)
		X.ERROR_ID := ID;
	ELSE
		IF X.STATE = BYTE#1 THEN (* Daten schreiben *)
			ra[1] := OSCAT_BASIC.REAL_TO_DW(X:=IN_REAL1);
			ra[2] := OSCAT_BASIC.REAL_TO_DW(X:=IN_REAL2);
			ra[3] := DINT_TO_DWORD(IN_DINT1);
			ra[4] := DINT_TO_DWORD(IN_DINT2);
			ra[5] := UDINT_TO_DWORD(IN_UDINT1);
			ra[6] := UDINT_TO_DWORD(IN_UDINT2);
			ra[7] := IN_DWORD1;
			ra[8] := IN_DWORD2;
			X.S_BUF.BUFFER[index] := ID; (* ID *)
			index := index + 1;
			X.S_BUF.BUFFER[index] := BYTE#21; (* TYPE X8 *)
			index := index + 1;
			FOR i2 := 1 TO 8 DO;
				FOR i := 1 TO 4 DO;
					X.S_BUF.BUFFER[index] := DWORD_TO_BYTE(ra[i2]);
					ra[i2] := ROR(ra[i2],8);
					index := index + 1;
				END_FOR;
			END_FOR;

		ELSIF X.STATE = BYTE#2 THEN (* Daten lesen *)
			index2 := index + 1; (* PCWORX Workaround *)
			IF X.R_BUF.BUFFER[index] <> ID OR X.R_BUF.BUFFER[index2] <> BYTE#21 THEN (* TYPE X8 *)
				X.ERROR_ID := ID;
			ELSE
				index := index + 2;
				FOR i2 := 1 TO 8 DO;
					ra[i2] := DWORD#0;
					FOR i := 1 TO 4 DO;
						ra[i2] := ra[i2] OR BYTE_TO_DWORD(X.R_BUF.BUFFER[index]);
						ra[i2] := ROR(ra[i2],8);
						index := index + 1;
					END_FOR;
				END_FOR;
				OUT_REAL1 := OSCAT_BASIC.DW_TO_REAL(X:=ra[1]);
				OUT_REAL2 := OSCAT_BASIC.DW_TO_REAL(X:=ra[2]);
				OUT_DINT1 := DWORD_TO_DINT(ra[3]);
				OUT_DINT2 := DWORD_TO_DINT(ra[4]);
				OUT_UDINT1 := DWORD_TO_UDINT(ra[5]);
				OUT_UDINT2 := DWORD_TO_UDINT(ra[6]);
				OUT_DWORD1 := ra[7];
				OUT_DWORD2 := ra[8];
			END_IF;
		END_IF;
		X.index := index;
	END_IF;
END_IF;

(* revision history
ks	15.may. 2011	rev 1.0
	original version

*)

END_FUNCTION_BLOCK

// POUs/OTHER/NETWORK_VERSION
FUNCTION NETWORK_VERSION : DWORD
VAR_INPUT
	IN : BOOL;
END_VAR

(*
version 1.0	02. feb 2011
programmer 	kst
tested by		oscat

network_version returns the version number in dword format
110 is library version 1.10
if IN = true, the release date will be returned

*)

IF in THEN
	NETWORK_VERSION := DATE_TO_DWORD(D#2012-12-31);
ELSE
	NETWORK_VERSION := 130;
END_IF;

(* revision history
ks	2. feb 2011	rev 1.0
	original version

*)

END_FUNCTION

// POUs/CONVERT/RC4_CRYPT_STREAM
FUNCTION_BLOCK RC4_CRYPT_STREAM
VAR_IN_OUT
	MODE : INT;
	KEY : STRING(40);
	BUF : ARRAY [0..63] OF BYTE;
	SIZE : UDINT;
END_VAR

VAR_OUTPUT
	POS : UDINT;
END_VAR

VAR
	sbox : ARRAY [0..255] OF BYTE;
	skey : ARRAY [0..255] OF BYTE;
	a : INT;
	b : INT;
	c : INT;
	d : USINT;
	e : USINT;
	end : UDINT;
	v : BYTE;
END_VAR

(*
version 1.0	09. jan. 2010
programmer	ks
tested BY	ks

RC4_CRYPT_STREAM kann einen Datenstrom ver/entschlüsseln mittels der RC4 Stromchiffrierung
*)

CASE MODE OF

1:	(* Initialisierung *)
	b := LEN(KEY) - 1;
	IF b < 0 OR SIZE < 1 THEN
		MODE := 3;
		RETURN;
	END_IF;

	FOR a := 0 TO b DO
		skey[a] := OSCAT_BASIC.CODE(KEY, a + 1);
		sbox[a] := INT_TO_BYTE(a);
	END_FOR;

	c := 0;
	FOR a := b + 1 TO 255 DO
		skey[a] := skey[c];
		sbox[a] := INT_TO_BYTE(a);
		c := c + 1;
		IF c > b THEN c := 0; END_IF;
	END_FOR;

	d := 0;
	FOR a := 0 TO 255 DO
		d := d + sbox[a] + skey[a];
		v := sbox[a];
		sbox[a] := sbox[d];
		sbox[d] := v;
	END_FOR;

	POS := 0;
	end := SIZE;
	SIZE := MIN(64,end);
	d := 0;
	e := 0;
	MODE := 2;

2:	(* Daten ver/entschlüsseln *)

	b := UDINT_TO_INT(SIZE) - 1;
	FOR a := 0 TO b DO
		d := d + 1;
		e := e + sbox[d];
		v := sbox[d];
		sbox[d] := sbox[e];
		sbox[e] := v;
		v := sbox[d] + sbox[e];
		BUF[a] :=BUF[a] XOR sbox[v];
	END_FOR;

	POS := POS + SIZE;
	SIZE := MIN(64,end - POS);

	IF SIZE = 0 THEN
		MODE := 3;
	END_IF;
END_CASE;

(* revision history

ks	9. Jan. 2010 rev 1.0
	original version

*)

END_FUNCTION_BLOCK

// POUs/CONVERT/SHA1_STR
FUNCTION_BLOCK SHA1_STR
VAR_INPUT
	RUN: BOOL;
END_VAR
VAR_OUTPUT
	DONE: BOOL;
END_VAR
VAR_IN_OUT
	STR: STRING(OSCAT_BASIC.STRING_LENGTH);
	SHA1 : ARRAY [0..19] OF BYTE;
END_VAR

VAR
	run_last: BOOL;
	SHA1_STREAM : SHA1_STREAM;
	buf : ARRAY [0..63] OF BYTE;
	mode : INT;
	size : UDINT;
	pos : UDINT;
END_VAR

(*
version 1.0	06. dec. 2009
programmer 	ks
tested BY	ks

SHA1_STR berechnet den MD5 Hash eines Strings
*)

CASE mode OF
0:	(* Wait für Start *)
	IF RUN AND NOT run_last THEN
		DONE := FALSE;
		mode := 1; (* Initialisierung *)
		size := LEN(STR);
	END_IF;

2:	(* Data copy and Calc *)
	IF size > 0 THEN
		OSCAT_BASIC._STRING_TO_BUFFER(STR:=MID(STR, UDINT_TO_INT(SIZE), UDINT_TO_INT(POS) + 1), POS:=0, PT:=ADR(buf), SIZE:=SIZEOF(buf));
	END_IF;

3:	DONE := TRUE;
	mode := 0; (* Stop *)

END_CASE;

IF mode > 0 THEN
	SHA1_STREAM(SIZE:=size, MODE:=mode, BUF:=buf, SHA1:=SHA1, POS=>pos);
END_IF;

run_last := RUN;

(* revision history

ks	6. dec. 2009 rev 1.0
	original version

*)

END_FUNCTION_BLOCK

// POUs/CONVERT/SHA1_TO_STRH
FUNCTION SHA1_TO_STRH : STRING(40)
VAR_INPUT
	SHA1 : ARRAY [0..19] OF BYTE;
END_VAR
VAR
	i : INT;
	tmp : BYTE;
	pt : POINTER TO BYTE;
END_VAR
(*
version 1.1	03. dec. 2011
programmer 	ks
tested BY	ks

SHA1_TO_STRH konvertiert das SHA1 Hash Array in einen HEX-String
*)

pt := ADR(SHA1_TO_STRH); (* read output adress to pointer *)

FOR i := 0 TO 19 DO; (* write the 10 hex characters backwards *)
	tmp := SHR(SHA1[i],4);
	PT^ := tmp + SEL(tmp <= 9,87,48);
	pt := pt + 1; (* decrement the pointer *)
	tmp := SHA1[i] AND 2#1111;
	PT^ := tmp + SEL(tmp <= 9,87,48);
	pt := pt + 1; (* decrement the pointer *)
END_FOR;
pt^:= 0; (* write the closing byte for the string *)

(* revision history

ks	6. dec. 2009 rev 1.0
	original version

ks	3. dec. 2011 rev 1.1
	incorrect string size
*)

END_FUNCTION

// POUs/NETWORK/SNTP_CLIENT
FUNCTION_BLOCK SNTP_CLIENT
VAR_IN_OUT
	IP_C : IP_C; (* IP_Control Verwaltungsstruktur *)
	S_BUF : NETWORK_BUFFER;
	R_BUF : NETWORK_BUFFER;
END_VAR
VAR_INPUT
	IP4 : DWORD;
	ACTIVATE : BOOL;
END_VAR
VAR_OUTPUT
	ERROR : DWORD;
	DONE_P : BOOL;
	UDT : DT;
	XMS : INT;
END_VAR
VAR
	IP_FIFO : IP_FIFO;
	ip_state : BYTE;
	ip_id : BYTE;
	i : INT;
	last : DWORD;
	state : INT;
	tx : DWORD;
	activate_last : BOOL;
	ip4_stored : DWORD;

	(*LOG_MSG : LOG_MSG;
	_debug_enable : BOOL := TRUE;*)

END_VAR

(*
version 1.1		20. oct. 2009
programmer 		ks
tested by		ks

SNTP_CLIENT führt eine SNTP-Anfrage bei einem SNTP/NTP-Server um die aktuelle Uhrzeit zu erhalten
*)

(* Domain Name System (query) *)
tx := OSCAT_BASIC.T_PLC_MS(); (* read system time *)

CASE state OF
00: (* auf positive Flanke SET warten *)
	DONE_P := FALSE;
	IF ACTIVATE AND NOT activate_last THEN
		ip4_stored := IP4; (* aktuelle IP4 speichern *)
		state := 10;
		ERROR := DWORD#0;
		ip_state := BYTE#1; (* Anmelden *)
		(*####################  DEBUG-MESSAGE  ###################################*)
		(*IF _debug_enable THEN
			LOG_CL.NEW_MSG := 'SNTP: S00 START';
			LOG_MSG();
		END_IF;*)
		(*########################################################################*)
	END_IF;

10: (* Bei IP_Control anmelden und auf freigabe warten *)
	IF ip_state = BYTE#3 THEN

		S_BUF.BUFFER[00] := BYTE#16#1B;
		FOR i := 1 TO 47 DO
			S_BUF.BUFFER[i] := BYTE#16#00;
		END_FOR;

		last := tx; (* aktuellen time wert sichern *)
		state := 30;

		(* IP Datenverkehr einrichten *)
		IP_C.C_PORT := WORD#123; (* Portnummer eintragen *)
		IP_C.C_IP := ip4_stored; (* IP eintragen *)
		IP_C.C_MODE := BYTE#1; (* Mode: UDP+AKTIV+PORT+IP *)
		IP_C.C_ENABLE := TRUE; (* Verbindungsaufbau freigeben *)
		IP_C.TIME_RESET := TRUE; (* Zeitueberwachung rücksetzen *)
		IP_C.R_OBSERVE := TRUE; (* Datenempfang ueberwachen *)
		S_BUF.SIZE := UINT#48; (* Sendelänge eintragen *)
		R_BUF.SIZE := UINT#0; (* Empfangslänge rücksetzen *)
    		(*####################  DEBUG-MESSAGE  ###################################*)
    		(*IF _debug_enable THEN
      			LOG_CL.NEW_MSG := 'SNTP: S10 SEND';
      			LOG_MSG();
    		END_IF;*)
    		(*########################################################################*)
	END_IF;

30:
	IF IP_C.ERROR <> DWORD#00 THEN
		ERROR := IP_C.ERROR;
		S_BUF.SIZE := UINT#0;
		R_BUF.SIZE := UINT#0;
		state := 0;
    		(*####################  DEBUG-MESSAGE  ###################################*)
    		(*IF _debug_enable THEN
      			LOG_CL.NEW_MSG := 'SNTP: S30 ERROR ~1';
      			LOG_CL.PRINTF[1] := DWORD_TO_STRING(ERROR);
      			LOG_MSG();
    		END_IF;*)
    		(*########################################################################*)

	ELSIF S_BUF.SIZE = UINT#0 AND R_BUF.SIZE >= UINT#48 THEN (* länge der empfangenen Daten prüfen *)

		(* Umrechnung SNTP Timestamp Base 1900-01-01 -> Unix 1970-01-01 = +2208988800 sekunden*)
		UDT := DWORD_TO_DT(OSCAT_BASIC.DWORD_OF_BYTE(R_BUF.BUFFER[40],R_BUF.BUFFER[41],R_BUF.BUFFER[42],R_BUF.BUFFER[43]) - DWORD#2208988800);

		(* Original-Sekundenanteile sind als 32 Bit Fractal dargestellt *)
		(* ms nur mit veringerte Auflösung berechnen 1/65535 -> Highword verwenden *)
		XMS := DWORD_TO_INT(SHR(DINT_TO_DWORD(WORD_TO_DINT(OSCAT_BASIC.WORD_OF_BYTE(R_BUF.BUFFER[44],R_BUF.BUFFER[45])) * DINT#1000),16));
		(* Zeitdifferenz (Laufzeitfehler) zwischen Send und Receive /2 teilen und addieren *)
		XMS := XMS + DWORD_TO_INT(SHR(tx - last,1));

		UDT := DWORD_TO_DT(DT_TO_DWORD(UDT) + (XMS / 1000)); (* sekundenanteile der Zeitdifferenz zu UDT aufrechnen *)
		XMS := XMS MOD 1000;  (* ms übernehmen *)
		state := 0;
		DONE_P := TRUE;
    		(*####################  DEBUG-MESSAGE  ###################################*)
    		(*IF _debug_enable THEN
        			LOG_CL.NEW_MSG := 'SNTP: S30 OK';
        			LOG_MSG();
    		END_IF;*)
    		(*########################################################################*)

	END_IF;

	IF state = 0 THEN
		IP_C.R_OBSERVE := FALSE; (* Datenempfang ueberwachen *)
		ip_state := BYTE#4;
	END_IF;

END_CASE;

activate_last := ACTIVATE; (* letzten Status sichern zur Flankenerkennung *)

(* IP_FIFO *)
IP_FIFO(FIFO:=IP_C.FIFO,STATE:=ip_state,ID:=ip_id);

(* revision history
ks	18. oct. 2008	rev 1.0
	original version

ks	20. oct. 2009	rev 1.1
	Networkbuffer und Buffer-funktionen auf Basis 0

*)

(***************************************************************************************)
(*               SNTP Datenstruktur
                                  1                   2                   3   
              0 1 2 3 4 5 6 7 8 9 0 1 2 3 4 5 6 7 8 9 0 1 2 3 4 5 6 7 8 9 0 1 
             +-+-+-+-+-+-+-+-+-+-+-+-+-+-+-+-+-+-+-+-+-+-+-+-+-+-+-+-+-+-+-+-+
Byte: 01-04  |LI | VN  |Mode |    Stratum    |     Poll      |   Precision   |
             +-+-+-+-+-+-+-+-+-+-+-+-+-+-+-+-+-+-+-+-+-+-+-+-+-+-+-+-+-+-+-+-+
Byte: 05-08  |                          Root  Delay (32 Bit)                 |
             +-+-+-+-+-+-+-+-+-+-+-+-+-+-+-+-+-+-+-+-+-+-+-+-+-+-+-+-+-+-+-+-+
Byte: 09-12  |                       Root  Dispersion (32 Bit)               |
             +-+-+-+-+-+-+-+-+-+-+-+-+-+-+-+-+-+-+-+-+-+-+-+-+-+-+-+-+-+-+-+-+
Byte: 13-16  |                     Reference Identifier (32 Bit)             |
             +-+-+-+-+-+-+-+-+-+-+-+-+-+-+-+-+-+-+-+-+-+-+-+-+-+-+-+-+-+-+-+-+
Byte: 17-24  |                    Reference Timestamp (64 Bit)               |
             +-+-+-+-+-+-+-+-+-+-+-+-+-+-+-+-+-+-+-+-+-+-+-+-+-+-+-+-+-+-+-+-+
Byte: 25-32  |                    Originate Timestamp (64 Bit)               |
             +-+-+-+-+-+-+-+-+-+-+-+-+-+-+-+-+-+-+-+-+-+-+-+-+-+-+-+-+-+-+-+-+
Byte: 33-40  |                     Receive Timestamp (64 Bit)                |
             +-+-+-+-+-+-+-+-+-+-+-+-+-+-+-+-+-+-+-+-+-+-+-+-+-+-+-+-+-+-+-+-+
Byte: 41-48  |                     Transmit Timestamp (64 Bit)               |
             +-+-+-+-+-+-+-+-+-+-+-+-+-+-+-+-+-+-+-+-+-+-+-+-+-+-+-+-+-+-+-+-+
Byte: 49-52  |                 Key Identifier (optional) (32 Bit)            |
             +-+-+-+-+-+-+-+-+-+-+-+-+-+-+-+-+-+-+-+-+-+-+-+-+-+-+-+-+-+-+-+-+
Byte: 53-68  |                 Message Digest (optional) (128 Bit)           |
             +-+-+-+-+-+-+-+-+-+-+-+-+-+-+-+-+-+-+-+-+-+-+-+-+-+-+-+-+-+-+-+-+

*)

(*
Worldwide NTP-Server


NIST-Zeitserver
• time-a.nist.gov
129.6.15.28 
NIST, Gaithersburg, Maryland 
• time-a.nist.gov
129.6.15.28 
NIST, Gaithersburg, Maryland 
• time-a.timefreq.bldrdoc.gov
132.163.4.101 (Stand: 1. Dezember 1999)
NIST, Boulder, Colorado 
• time-b.timefreq.bldrdoc.gov
132.163.4.102 (Stand: 1. Dezember 1999)
NIST, Boulder, Colorado 
• time-c.timefreq.bldrdoc.gov
132.163.4.103 (Stand: 1. Dezember 1999)
NIST, Boulder, Colorado 
• utcnist.colorado.edu
128.138.140.44
University of Colorado, Boulder 
• time.nist.gov
192.43.244.18
NCAR, Boulder, Colorado 
• time-nw.nist.gov
131.107.1.10
Microsoft, Redmond, Washington 
• nist1.dc.certifiedtime.com
216.200.93.8
Abovnet, North Virginia 
• nist1.datum.com
209.0.72.7
Datum, San Jose, Kalifornien 
• nist1.nyc.certifiedtime.com
208.184.49.129 
Abovnet, New York City 
• nist1.sjc.certifiedtime.com
207.126.103.202
Abovnet, San Jose, Kalifornien 

Zeitserver der ersten Ebene
Sortiert nach Standort: 
Nordamerika
• Palo Alto, Kalifornien: Systems Research Center, Compaq Computer Corp.
204.123.2.72: usno.pa-x.dec.com; CNAME: navobs1.pa-x.dec.com
Servicebereich: US-Zeitzonen PST (Pacific Standard Time) und MST (Mountain Standard Time) 
• Marina del Rey, Kalifornien: USC Information Sciences Institute
128.9.176.30: timekeeper.isi.edu
Servicebereich: CalRen2- und Los Nettos-Bereich  
• Washington, DC: U.S. Naval Observatory
192.5.41.41: tock.usno.navy.mil 
192.5.41.40: tick.usno.navy.mil
Servicebereich: NSFNET 
• Ottawa, Ontario, Kanada: National Research Council of Canada
time.chu.nrc.ca
Servicebereich: Kanada 
• Raleigh, North Carolina: North Carolina State University
152.1.58.124: terrapin.csc.ncsu.edu
Servicebereich: Südosten der USA 
• Cambridge, Massachusetts: MIT Information Systems
18.72.0.3: bitsy.mit.edu 
Servicebereich: NSFNET- und NEARnet-Bereich 
• Cambridge, Massachusetts: MIT
18.26.4.105: bonehed.lcs.mit.edu
Servicebereich: Osten der USA 
• Palo Alto, Kalifornien: Internet Software Consortium
192.5.5.250: clock.isc.org
Servicebereich: BARRnet, Alternet-West und CIX-West 
• Cambridge, Massachusetts: Open Software Foundation
130.105.4.59: clock.osf.org
Servicebereich: NSFNET- und NEARnet-Bereich 
• Palo Alto, Kalifornien: ViaNet Communications
209.81.9.7: clock.via.net 
• Cleveland, Ohio: Lewis Research Center (NASA)
128.156.1.43: lerc-dns.lerc.nasa.gov
Servicebereich: NSFNET und OARNET 
• Colorado Springs, Colorado: Schriever AFB
204.34.198.40: navobs1.usnogps.navy.mil; CNAME: tick.usnogps.navy.mil 
204.34.198.41: navobs1.usnogps.navy.mil; CNAME: tock.usnogps.navy.mil 
Servicebereich: US-Zeitzonen PST (Pacific Standard Time) und MST (Mountain Standard Time) 
• St. Louis, Missouri: Washington University
128.252.19.1: navobs1.usnogps.navy.mil; CNAME: tick.wustl.edu 
Servicebereich: US-Zeitzone CST (Central Standard Time) 
• Research Triangle Park, North Carolina: MCNC
192.101.21.1: ncnoc.ncren.net
Servicebereich: NC-REN-Bereich (North Carolina Research and Education Network) 
• Cupertino, Kalifornien: HP
192.6.38.127: ntp-cup.external.hp.com
Servicebereich: USA Westküste 
• Newark, Delaware: Conectiv Communications
138.39.7.20: ntp1.delmarva.com
Servicebereich: Cable & Wireless Network (früher MCInet) 
• University Park, Pennsylvania: Penn State University
128.118.46.3: otc1.psu.edu
Servicebereich: NSFNET, PREPNET und JvNCnet  

Europa
• Borowiec, Polen: Astrogeodynamical Observatory, Space Research Centre
150.254.183.15: vega.cbk.poznan.pl
Servicebereich: Polen und Europa 
• Stockholm, Schweden: Stupi AB
192.36.143.151: Time2.Stupi.SE
Servicebereich: Europa 
• Turin, Italien: IEN Galileo Ferraris
193.204.114.1: time.ien.it
Servicebereich: Italien und Europa 
• Zürich, Schweiz: Integrated Systems Laboratory , Eidgenössischen Technischen Hochschule Zürich 
129.132.2.21: swisstime.ethz.ch
Servicebereich: Schweiz und Europa 
• Turin, Italien: CSTV of National Research Council
150.145.33.1: tempo.cstv.to.cnr.it
Servicebereich: Italien und Europa 
• Erlangen, Deutschland: Universität Erlangen-Nürnberg
ntp0.fau.de; ntp1.fau.de; ntp2.fau.de; 
ntps1-0.uni-erlangen.de; ntps1-1.uni-erlangen.de; ntps1-2.uni-erlangen.de
Servicebereich: Deutschland und Europa 
• Berlin, Deutschland: Technische Universität Berlin
130.149.17.21: ntps1-0.cs.tu-berlin.de
130.149.17.8: ntps1-1.cs.tu-berlin.de
Servicebereich: Deutschland und Europa 
• Deutschland
131.173.17.7: ntps1-1.rz.Uni-Osnabrueck.DE
Servicebereich: Deutschland und Europa 
• Schweden
192.36.143.150: Time1.Stupi.SE
Servicebereich: SUnet und NORDUnet Schweden 

Fernost und pazifische Randgebiete
• Hong Kong: Chinesische Universität von Hong Kong. 
137.189.6.18: clock.cuhk.edu.hk
Servicebereich: Hong Kong (China) und Südostasien  
• Fukuoka, Japan: Universität Fukuoka
133.100.9.2: clock.nc.fukuoka-u.ac.jp
133.100.11.8: clock.tl.fukuoka-u.ac.jp
Servicebereich: Japan und pazifischer Raum  

Australien
• Melbourne, Australien: University of Melbourne
128.250.36.2: ntp.cs.mu.OZ.AU
Servicebereich: Australien und Neuseeland  

Zeitserver der zweiten Ebene
Nach geographischem Standort sortiert: 
Nordamerika
NTP-Zeitserver: • Quebec, Kanada: Canadian Meteorological Center
ntp1.cmc.ec.gc.ca; ntp2.cmc.ec.gc.ca 
Servicebereich: Ostkanada  
• Ontario, Kanada: National Research Council of Canada
time.chu.nrc.ca; time.nrc.ca
Servicebereich: Kanada 
• Saskatchewan, Kanada: University of Regina 
142.3.100.15: timelord.uregina.ca
Servicebereich: Kanada 
• Ontario, Kanada: University of Toronto
tick.utoronto.ca; tock.utoronto.ca
Servicebereich: Ostkanada  
• Mexiko: Audiotel-Büro 
ntp2a.audiotel.com.mx; ntp2c.audiotel.com.mx; ntp2b.audiotel.com.mx
Servicebereich: Avantel, MCINet und Mexiko 
• Santa Cruz, Kalifornien: Scruz-net, inc.
165.227.1.1: ns.scruz.net
Servicebereich: Westen der USA 
• San Diego, Kalifornien: UCSD Academic Computing Services/Network Operations
132.239.254.49: ntp.ucsd.edu
Servicebereich: CERFNET; NSFNET, SDSC-Bereich, und nahegelegene Bereiche 
• Quincy, Kalifornien 
ntp1.mainecoon.com; ntp2.mainecoon.com 
Servicebereich: Nordamerika 
• Newark, Delaware: University of Delaware
128.175.1.3: louie.udel.edu
Servicebereich: CAIRN, Abilene und vBNS  
• Atlanta, Georgia: CNSG
ntp.shorty.com
Servicebereich: Südwesten der USA  
• Kennesaw, Georgia: PeachNet 
rolex.peachnet.edu; timex.peachnet.edu
Servicebereich: PeachNet (Georgia) und Südwesten der USA  
• Urbana-Champaign, Illinois: University of Illinois
ntp-0.cso.uiuc.edu; ntp-1.cso.uiuc.edu; ntp-2.cso.uiuc.edu
Servicebereich: CICNET, Mittlerer Westen und NCSA-Bereich  
• Chicago, Illinois: Argonne National Laboratory 
ntp-1.mcs.anl.gov; ntp-2.mcs.anl.gov
Servicebereich: NSF/ANSNet, CICNet, NetIllinois und ESNet  
• West Lafayette, Indiana: Purdue University
gilbreth.ecn.purdue.edu; harbor.ecn.purdue.edu; molecule.ecn.purdue.edu 
Servicebereich: NSFNET- und CICNET-Bereich  
• Manhattan, Kansas: KansasNet OnLine Services
199.240.130.1: ntp1.kansas.net
199.240.130.12: ntp2.kansas.net
Servicebereich: Zentral-USA und Great Plains  
• Boston, Massachusetts: UMass-Boston CS dept.
158.121.104.4: timeserver.cs.umb.edu
Servicebereich: Neuengland  
• Minneapolis/St Paul, Minnesota: University of Minnesota
ns.nts.umn.edu; nss.nts.umn.edu
Servicebereich: CICNET-Bereich  
• Columbia, Missouri: University of Missouri-Columbia
128.206.206.12: everest.cclabs.missouri.edu
Servicebereich: MOREnet  
• Omaha, Nebraska: Radiks Internet Access
205.138.126.83: allison.radiks.net
Servicebereich: Mittlerer Westen, USA  
• Las Vegas, Nevada: University of Nevada System Computing Services
131.216.1.101: cuckoo.nevada.edu 
Servicebereich: NevadaNet, NSFNET und SDSC-Bereich  
• Las Vegas, Nevada: UNLV College of Engineering
tick.cs.unlv.edu; tock.cs.unlv.edu
Servicebereich: Sprintnet  
• New York City, New York: Columbia University
ntp.ctr.columbia.edu 
Servicebereich: Sprintlink und NYSERnet  
• Ithaca, New York: Cornell University 
192.35.82.50: ntp0.cornell.edu
Servicebereich: NSFNET und NYSER-Bereich  
• New York, New York: Morningside Campus, Columbia University
sundial.columbia.edu
Servicebereich: NYSERnet  
• New York City, New York: Columbia University Computer Science Department
timex.cs.columbia.edu 
Servicebereich: PSINET; NSFNET, und NYSER-Bereich  
• Norman, Oklahoma: University of Oklahoma
129.15.22.8: constellation.ecn.uoknor.edu 
Servicebereich: Midnet  
• Coos Bay, Oregon: Koala Computers
207.48.109.6: tick.koalas.com
Servicebereich: Nordwesten der USA  
• University Park, Pennsylvania: Penn State University
128.118.25.3: clock.psu.edu
Servicebereich: Internet2, vBNS, CERFnet(AT&T IP Services), PSC/NCNE und CASC 
• Pittsburgh, Pennsylvania: Pittsburgh Supercomputing Center
128.182.58.100: fuzz.psc.edu
Servicebereich: NSFNET und PSC-Bereich  
• Pittsburgh, Pennsylvania: Carnegie Mellon Electrical and Computer Engineering 
ntp-1.ece.cmu.edu; ntp-2.ece.cmu.edu 
Servicebereich: PREPNET und PSC-Bereich  
• Dallas, Texas: Cox School of Business, Southern Methodist University
129.119.80.126: ntp.cox.smu.edu 
Servicebereich: NSFNET und SESQUI-Bereich  
• Hughes Springs, Texas: First National Bank
209.144.20.76: ntp.fnbhs.com
Servicebereich: Nordosten Texas  
• Houston, Texas: Baylor College of Medicine
128.249.1.10: ntp.tmc.edu 
Servicebereich: NSFNET und SESQUI-Bereich  
• College Station, Texas: Texas A&M University
165.91.52.110: ntp5.tamu.edu
Servicebereich: NSFNET, SESQUI-Bereich, THEnet und TAMUSDSN 
• Plano, Texas: Greyware Automation Products
tick.greyware.com; tock.greyware.com
Servicebereich: Südzentral-USA  
• Blacksburg, Virginia: Virginia Tech Computing Center
ntp-1.vt.edu; ntp-2.vt.edu
Servicebereich: Südwesten der USA  
• Arlington, Virginia: Center for Seismic Studies
140.162.1.3: ntp.cmr.gov
Servicebereich: NSFNET und SURA-Bereich  
• Richland, Washington: Washington State University 
192.31.216.30: clock.tricity.wsu.edu
Servicebereich: NSFNET und NorthWestNet  
• Washington, USA: Mill Creek
time.ultimeth.net
Servicebereich: Nordwesten der USA  
• Wisconsin, USA: Computer Science Department, University of Wisconsin-Madison
ntp1.cs.wisc.edu; ntp2.cs.wisc.edu; ntp3.cs.wisc.edu
Servicebereich: USA und jeder andere  

Südamerika
• Buenos Aires, Argentinien: Network Access Point
200.49.40.1: CNAME: tick.nap.com.ar
200.49.32.1: CNAME: tock.nap.com.ar
Servicebereich: Argentinien 
• Buenos Aires, Argentinien: Sinectis S.A.
time.sinectis.com.ar 
Servicebereich: Argentinien 
• Brasilien: Brazilian Research Network
200.144.121.33: ntp.cais.rnp.br 
Servicebereich: Brasilien 
• Venezuela: VELUG, Grupo de Usuarios Linux de Venezuela
150.185.192.250: ntp.linux.org.ve
Servicebereich: Arica  

Europa
• Zürich, Schweiz: Eidgenössischen Technischen Hochschule Zürich
129.132.98.11: bernina.ethz.ch
Servicebereich: Schweiz und Europa  
• Standort: Kopenhagen, Dänemark, Europa 
clock.netcetera.dk; clock2.netcetera.dk 
Servicebereich: Dänemark, Skandinavien und Nordeuropa  
• Spanien: Altea 
slug.ctv.es
Servicebereich: Spanien  
• Pieksamaki, Finnland: Keski-Savon Oppimiskeskus
tick.keso.fi; tock.keso.fi
Servicebereich: Finnland  
• Meudon, Frankreich: Observatoire de Paris-Meudon 
ntp.obspm.fr 
Servicebereich: Frankreich und Europa  
• Lyon, Frankreich: CISM 
ntp.univ-lyon1.fr 
Servicebereich: Frankreich, Schweiz, Italien und Europa  
• Paris, Frankreich: VIA, Ecole Centrale
138.195.130.70: ntp.via.ecp.fr
Servicebereich: Frankreich und Europa  
• Budapest, Ungarn: KFKI Research Institute for Particle and Nuclear Physics
148.6.0.1: time.kfki.hu
Servicebereich: HUNGARNET  
• Italien: Net4u Srl, Vercelli, Italien
195.32.52.129: ntps.net4u.it
Servicebereich: Italien  
• Oslo, Norwegen: Universität Oslo
129.240.64.3: fartein.ifi.uio.no 
Servicebereich: NORDUnet  
• Oslo, Norwegen: Alcanet International
time.alcanet.no
Servicebereich: Europa 
• Krakau, Polen: Academic Computer Centre 
149.156.4.11: info.cyf-kr.edu.pl
Servicebereich: Polen und Europa  
• Lund, Schweden: Lund Institute of Technology
130.235.20.3: ntp.lth.se 
Servicebereich: Schweden und NORDUnet 
• Ljubljana, Slowenien: Institute of Biophysics, University of Ljubljana
biofiz.mf.uni-lj.si 193.2.69.11
Servicebereich: Slowenien und Europa  
• Ljubljana, Slowenien: Hydrometeorological Institute of Slovenia
hmljhp.rzs-hm.si
Servicebereich: Slowenien und Europa  
• Ljubljana, Slowenien: Academic and Research Network of Slovenia
ntp1.arnes.si; ntp2.arnes.si
Servicebereich: Slowenien und Europa  
• Ljubljana, Slowenien: J. Stefan Institute
time.ijs.si
Servicebereich: Slowenien und Europa  

Britische Inseln
• Dublin, Irland: School of Mathematics, Trinity College 
ntp.cs.tcd.ie; ntp.maths.tcd.ie; ntp.tcd.ie
Servicebereich: Irland und Großbritannien 
• Glasgow, Schottland: Strathclyde University 
ntp.cs.strath.ac.uk 
Servicebereich: Großbritannien, Europa und andere 
• Cambridge, Großbritannien
ntp0.uk.uu.net; ntp1.uk.uu.net; 
ntp2.uk.uu.net 
Servicebereich: UUNET (in Großbritannien früher auch als PIPEX bekannt) und Großbritannien.  
• Manchester, England: University of Manchester
ntp2a.mcc.ac.uk; ntp2b.mcc.ac.uk;
ntp2c.mcc.ac.uk; ntp2d.mcc.ac.uk 
Servicebereich: Großbritannien  
• Buckinghamshire, Großbritannien: Wibble U.K., Aylesbury
tick.tanac.net
Servicebereich: Großbritannien  

Asien
• Moskau, Russland: Landau Institute for Theoretical Physics
193.233.9.7: ntp.landau.ac.ru
Servicebereich: Russland  
• Russland: Pushchino (bei Moskau)
194.149.67.130: ntp.psn.ru
Servicebereich: Russland 
• Chernogolovka, Russland: Chernogolovka Scientific Center (bei Moskau)
193.233.46.10: sign.chg.ru
Servicebereich: Russland  

Fernost und pazifische Randgebiete
• Tokyo, Japan: Cyber Fleet, Inc.
203.139.30.195: ntp.cyber-fleet.net
Servicebereich: Japan und Ostasien  
• Seoul, Korea: Inet, Inc.
time.nuri.net
Servicebereich: Korea, Japan, Hong Kong und Ostasien  
• Hamilton, Neuseeland: Universität Waikato
truechimer.waikato.ac.nz; truechimer1.waikato.ac.nz; 
truechimer2.waikato.ac.nz; truechimer3.waikato.ac.nz
Servicebereich: Neuseeland  
• Singapur und Philippinen: 
ntp.shim.org 
Servicebereich: Singapur  

Afrika
• Lagos, Nigeria: Supernet300
ntp.supernet300.com
Servicebereich: Westafrika (hauptsächlich nigerischer NITEL-Backbone)  
• Pietermaritzburg, Südafrika: Natal University
143.128.82.200: ntp.cs.unp.ac.za
Servicebereich: Südafrika  

Australien
• Adelaide, Südaustralien: University of Adelaide
129.127.28.4: augean.eleceng.adelaide.edu.au
129.127.40.3: ntp.adelaide.edu.au
203.21.37.18: ntp.saard.net
Servicebereich: AARNet  
• Carlton, Victoria, Australien: eSec Limited
203.21.84.4: time.esec.com.au  

*)

END_FUNCTION_BLOCK

// POUs/NETWORK/SNTP_SERVER
FUNCTION_BLOCK SNTP_SERVER
VAR_IN_OUT
	IP_C : IP_C; (* IP_Control Verwaltungsstruktur *)
	S_BUF : NETWORK_BUFFER;
	R_BUF : NETWORK_BUFFER;
END_VAR
VAR_INPUT
	ENABLE : BOOL;
	STRATUM : BYTE := BYTE#1;
	UDT : DT;
	XMS : INT;
END_VAR
VAR
	IP_FIFO : IP_FIFO;
	ip_state : BYTE;
	ip_id : BYTE;
	i2 : INT;
	i : INT;
	timestamp_int : DWORD; (* Timestamp integer part *)
	timestamp_sek : DWORD; (* Timestamp fraction part (HIGH_WORD) *)
	ts_b : BYTE;
	state : INT;
	tx : UDINT;
	t : TON;

	(*LOG_MSG : LOG_MSG;
	_debug_enable : BOOL := TRUE;*)

END_VAR

(*
version 1.2		17. may. 2011
programmer 		ks
tested by			ks

SNTP_SERVER stellt Datum/Uhrzeit füR andere (S)NTP_CLIENTS zur Verfügung.
*)

(* Domain Name System (query) *)
tx := OSCAT_BASIC.T_PLC_MS(); (* read system time *)

CASE state OF

00: (* Warten auf Freigabe *)
	IF ENABLE THEN
		state := 10;
		ip_state := BYTE#1; (* Anmelden *)
    		(*####################  DEBUG-MESSAGE  ###################################*)
    		(*IF _debug_enable THEN
      			LOG_CL.NEW_MSG := 'SNTP_SERVER: S00 START';
      			LOG_MSG();
    		END_IF;*)
    		(*########################################################################*)
	END_IF;

10: (* Bei IP_Control anmelden und auf freigabe warten *)
	IF ip_state = BYTE#3 THEN
		(* IP Datenverkehr einrichten *)
		IP_C.C_PORT := WORD#123; (* Portnummer eintragen *)
		IP_C.C_IP := DWORD#00; (* IP eintragen *)
		IP_C.C_MODE := BYTE#5; (* Mode: UDP+PASSIV+PORT *)
		IP_C.C_ENABLE := TRUE; (* Verbindungsaufbau freigeben *)
		IP_C.TIME_RESET := TRUE; (* Zeitueberwachung rücksetzen *)
		IP_C.R_OBSERVE := FALSE; (* Datenempfang ueberwachen *)
		S_BUF.SIZE := UINT#0; (* Sendelänge eintragen *)
		R_BUF.SIZE := UINT#0; (* Empfangslänge rücksetzen *)
		state := 20;
    		(*####################  DEBUG-MESSAGE  ###################################*)
    		(*IF _debug_enable THEN
      			LOG_CL.NEW_MSG := 'SNTP_SERVER: S10 INIT';
      			LOG_MSG();
    		END_IF;*)
    		(*########################################################################*)
	END_IF;
20:
	IF R_BUF.SIZE > UINT#0 THEN
		state := 20;
    		(*####################  DEBUG-MESSAGE  ###################################*)
    		(*IF _debug_enable THEN
      			LOG_CL.NEW_MSG := 'SNTP_SERVER: S20 REQUEST - Size: ~1';
      			LOG_CL.PRINTF[1] := UINT_TO_STRING(R_BUF.SIZE);
      			LOG_MSG();
    		END_IF;*)
    		(*########################################################################*)
		(* empfangenes Telegramm mit 00 auffüllen , wenn zu kurz ! und Sendebuffer mit 00 vorbelegen *)
		FOR i := 0 TO 47 DO
			IF INT_TO_UINT(i) > R_BUF.SIZE - 1 THEN
				R_BUF.BUFFER[i] := BYTE#00;
			END_IF;
			S_BUF.BUFFER[i] := BYTE#00;
		END_FOR;

		R_BUF.SIZE := UINT#0;

		(* Sendedaten aufbereiten *)
		S_BUF.BUFFER[0] := BYTE#2#11100; (* Flags: NO WARNING, NTP VERSION 3 , SERVER *)
		S_BUF.BUFFER[1] := STRATUM; (* Peer Clock Stratum: *)
		S_BUF.BUFFER[2] := BYTE#10; (* Peer Polling Intervall 2 hoch 10 = 1024 sek. *)
		S_BUF.BUFFER[3] := BYTE#16#FB; (* Peer Clock Precision: -5 = -31,25ms *)

		(* Umrechnung SNTP Timestamp Base 1900-01-01 = Unix 1970-01-01 + 2208988800 sekunden *)
		timestamp_int := DT_TO_DWORD(UDT) + DWORD#2208988800;

		(* Sekundenanteile sind als 32 Bit Fractal dargestellt *)
		(* nur mit veringerte Auflösung berechnen 1/65535 -> Highword verwenden *)
		(* Berechnung des Sekundenanteils: xms * 65535 / 1000 *)
		timestamp_sek := DINT_TO_DWORD(DWORD_TO_DINT(SHL(INT_TO_DWORD(XMS),16))/DINT#1000);

		ts_b := OSCAT_BASIC.BYTE_OF_DWORD(timestamp_int,3); (* Timestamp Byte 3 *)
		S_BUF.BUFFER[16] := ts_b; (* Reference Timestamp *)
		S_BUF.BUFFER[32] := ts_b; (* Receive   Timestamp *)
		S_BUF.BUFFER[40] := ts_b; (* Transmit  Timestamp *)

		ts_b := OSCAT_BASIC.BYTE_OF_DWORD(TIMESTAMP_INT,2); (* Timestamp Byte 2 *)
		S_BUF.BUFFER[17] := ts_b; (* Reference Timestamp *)
		S_BUF.BUFFER[33] := ts_b; (* Receive   Timestamp *)
		S_BUF.BUFFER[41] := ts_b; (* Transmit  Timestamp *)

		ts_b := OSCAT_BASIC.BYTE_OF_DWORD(TIMESTAMP_INT,1); (* Timestamp Byte 1 *)
		S_BUF.BUFFER[18] := ts_b; (* Reference Timestamp *)
		S_BUF.BUFFER[34] := ts_b; (* Receive   Timestamp *)
		S_BUF.BUFFER[42] := ts_b; (* Transmit  Timestamp *)

